LIN {X 0,Y 422.722,Z 380.789,A -85,B 0,C 180,E1 -10186.884,E2 -10186.884} C_VEL
LIN {X 0,Y 423.061,Z 367.924,A -85,B 0,C 180,E1 -10187.181,E2 -10187.181} C_VEL
LIN {X 0,Y 423.842,Z 291.469,A -85,B 0,C 180,E1 -10188.511,E2 -10188.511} C_VEL
LIN {X 0,Y 419.727,Z 266.585,A -85,B 0,C 180,E1 -10189.181,E2 -10189.181} C_VEL
LIN {X 0,Y 420.786,Z 249.269,A -85,B 0,C 180,E1 -10192.591,E2 -10192.591} C_VEL
LIN {X 0,Y 421.199,Z 242.855,A -85,B 0,C 180,E1 -10193.868,E2 -10193.868} C_VEL
LIN {X 0,Y 419.611,Z 233.827,A -85,B 0,C 180,E1 -10195.815,E2 -10195.815} C_VEL
LIN {X 0,Y 418.321,Z 227.378,A -85,B 0,C 180,E1 -10197.293,E2 -10197.293} C_VEL
LIN {X 0,Y 418.246,Z 227.386,A -85,B 0,C 180,E1 -10200.272,E2 -10200.272} C_VEL
LIN {X 0,Y 418.249,Z 227.389,A -85,B 0,C 180,E1 -10203.677,E2 -10203.677} C_VEL
LIN {X 0,Y 418.239,Z 227.391,A -85,B 0,C 180,E1 -10207.224,E2 -10207.224} C_VEL
LIN {X 0,Y 418.247,Z 227.385,A -85,B 0,C 180,E1 -10209.682,E2 -10209.682} C_VEL
LIN {X 0,Y 418.232,Z 227.384,A -85,B 0,C 180,E1 -10212.321,E2 -10212.321} C_VEL
LIN {X 0,Y 418.238,Z 227.388,A -85,B 0,C 180,E1 -10215.109,E2 -10215.109} C_VEL
LIN {X 0,Y 418.24,Z 227.383,A -85,B 0,C 180,E1 -10217.767,E2 -10217.767} C_VEL
LIN {X 0,Y 418.249,Z 227.385,A -85,B 0,C 180,E1 -10220.62,E2 -10220.62} C_VEL
LIN {X 0,Y 418.244,Z 227.382,A -85,B 0,C 180,E1 -10223.976,E2 -10223.976} C_VEL
LIN {X 0,Y 418.257,Z 227.386,A -85,B 0,C 180,E1 -10227.156,E2 -10227.156} C_VEL
LIN {X 0,Y 418.268,Z 227.385,A -85,B 0,C 180,E1 -10230.895,E2 -10230.895} C_VEL
LIN {X 0,Y 418.27,Z 227.38,A -85,B 0,C 180,E1 -10234.096,E2 -10234.096} C_VEL
LIN {X 0,Y 418.237,Z 227.385,A -85,B 0,C 180,E1 -10237.264,E2 -10237.264} C_VEL
LIN {X 0,Y 418.283,Z 227.379,A -85,B 0,C 180,E1 -10240.364,E2 -10240.364} C_VEL
LIN {X 0,Y 418.316,Z 227.377,A -85,B 0,C 180,E1 -10243.405,E2 -10243.405} C_VEL
LIN {X 0,Y 418.346,Z 227.372,A -85,B 0,C 180,E1 -10246.999,E2 -10246.999} C_VEL
LIN {X 0,Y 418.34,Z 227.369,A -85,B 0,C 180,E1 -10250.329,E2 -10250.329} C_VEL
LIN {X 0,Y 418.486,Z 227.355,A -85,B 0,C 180,E1 -10253.249,E2 -10253.249} C_VEL
LIN {X 0,Y 418.338,Z 227.371,A -85,B 0,C 180,E1 -10255.182,E2 -10255.182} C_VEL
LIN {X 0,Y 418.544,Z 227.347,A -85,B 0,C 180,E1 -10258.076,E2 -10258.076} C_VEL
LIN {X 0,Y 418.67,Z 227.325,A -85,B 0,C 180,E1 -10260,E2 -10260} C_VEL
LIN {X 0,Y 418.508,Z 227.352,A -85,B 0,C 180,E1 -10262.888,E2 -10262.888} C_VEL
LIN {X 0,Y 418.49,Z 227.357,A -85,B 0,C 180,E1 -10266.751,E2 -10266.751} C_VEL
LIN {X 0,Y 418.4,Z 227.365,A -85,B 0,C 180,E1 -10268.695,E2 -10268.695} C_VEL
LIN {X 0,Y 418.315,Z 227.371,A -85,B 0,C 180,E1 -10271.631,E2 -10271.631} C_VEL
LIN {X 0,Y 418.303,Z 227.38,A -85,B 0,C 180,E1 -10274.597,E2 -10274.597} C_VEL
LIN {X 0,Y 418.287,Z 227.378,A -85,B 0,C 180,E1 -10277.604,E2 -10277.604} C_VEL
LIN {X 0,Y 418.25,Z 227.387,A -85,B 0,C 180,E1 -10280.663,E2 -10280.663} C_VEL
LIN {X 0,Y 418.274,Z 227.379,A -85,B 0,C 180,E1 -10283.782,E2 -10283.782} C_VEL
LIN {X 0,Y 418.266,Z 227.384,A -85,B 0,C 180,E1 -10287.059,E2 -10287.059} C_VEL
LIN {X 0,Y 418.242,Z 227.386,A -85,B 0,C 180,E1 -10290.273,E2 -10290.273} C_VEL
LIN {X 0,Y 418.247,Z 227.388,A -85,B 0,C 180,E1 -10293.678,E2 -10293.678} C_VEL
LIN {X 0,Y 418.234,Z 227.388,A -85,B 0,C 180,E1 -10297.225,E2 -10297.225} C_VEL
LIN {X 0,Y 418.208,Z 227.393,A -85,B 0,C 180,E1 -10300.868,E2 -10300.868} C_VEL
LIN {X 0,Y 418.263,Z 227.487,A -85,B 0,C 180,E1 -10301.906,E2 -10301.906} C_VEL
LIN {X 0,Y 420.256,Z 237.548,A -85,B 0,C 180,E1 -10304.212,E2 -10304.212} C_VEL
LIN {X 0,Y 420.082,Z 245.787,A -85,B 0,C 180,E1 -10305.915,E2 -10305.915} C_VEL
LIN {X 0,Y 424.209,Z 265.63,A -85,B 0,C 180,E1 -10306.479,E2 -10306.479} C_VEL
LIN {X 0,Y 422.976,Z 353.633,A -85,B 0,C 180,E1 -10308.027,E2 -10308.027} C_VEL
LIN {X 0,Y 422.598,Z 366.879,A -85,B 0,C 180,E1 -10308.46,E2 -10308.46} C_VEL
LIN {X 0,Y 422.118,Z 378.903,A -85,B 0,C 180,E1 -10309.037,E2 -10309.037} C_VEL
LIN {X 0,Y 421.52,Z 390.055,A -85,B 0,C 180,E1 -10309.752,E2 -10309.752} C_VEL
LIN {X 0,Y 420.847,Z 400.567,A -85,B 0,C 180,E1 -10310.611,E2 -10310.611} C_VEL
LIN {X 0,Y 420.062,Z 411.702,A -85,B 0,C 180,E1 -10311.754,E2 -10311.754} C_VEL
LIN {X 0,Y 419.343,Z 420.671,A -85,B 0,C 180,E1 -10312.89,E2 -10312.89} C_VEL
LIN {X 0,Y 418.81,Z 428.099,A -85,B 0,C 180,E1 -10314.032,E2 -10314.032} C_VEL
LIN {X 0,Y 418.248,Z 435.582,A -85,B 0,C 180,E1 -10315.424,E2 -10315.424} C_VEL
LIN {X 0,Y 417.798,Z 441.651,A -85,B 0,C 180,E1 -10316.825,E2 -10316.825} C_VEL
LIN {X 0,Y 417.439,Z 447.432,A -85,B 0,C 180,E1 -10318.539,E2 -10318.539} C_VEL
LIN {X 0,Y 417.213,Z 451.593,A -85,B 0,C 180,E1 -10320.203,E2 -10320.203} C_VEL
LIN {X 0,Y 416.996,Z 454.414,A -85,B 0,C 180,E1 -10321.842,E2 -10321.842} C_VEL
LIN {X 0,Y 416.848,Z 455.921,A -85,B 0,C 180,E1 -10323.326,E2 -10323.326} C_VEL
LIN {X 0,Y 416.819,Z 456.5,A -85,B 0,C 180,E1 -10325.069,E2 -10325.069} C_VEL
LIN {X 0,Y 416.839,Z 456.196,A -85,B 0,C 180,E1 -10326.131,E2 -10326.131} C_VEL
LIN {X 0,Y 416.934,Z 454.562,A -85,B 0,C 180,E1 -10327.988,E2 -10327.988} C_VEL
LIN {X 0,Y 417.183,Z 451.479,A -85,B 0,C 180,E1 -10329.797,E2 -10329.797} C_VEL
LIN {X 0,Y 417.412,Z 447.619,A -85,B 0,C 180,E1 -10331.343,E2 -10331.343} C_VEL
LIN {X 0,Y 417.656,Z 442.562,A -85,B 0,C 180,E1 -10332.874,E2 -10332.874} C_VEL
LIN {X 0,Y 418.107,Z 436.133,A -85,B 0,C 180,E1 -10334.398,E2 -10334.398} C_VEL
LIN {X 0,Y 418.655,Z 428.087,A -85,B 0,C 180,E1 -10335.912,E2 -10335.912} C_VEL
LIN {X 0,Y 419.285,Z 419.45,A -85,B 0,C 180,E1 -10337.215,E2 -10337.215} C_VEL
LIN {X 0,Y 420.006,Z 409.662,A -85,B 0,C 180,E1 -10338.416,E2 -10338.416} C_VEL
LIN {X 0,Y 420.695,Z 398.721,A -85,B 0,C 180,E1 -10339.496,E2 -10339.496} C_VEL
LIN {X 0,Y 420.832,Z 397.065,A -85,B 0,C 180,E1 -10339.634,E2 -10339.634} C_VEL
LIN {X 0,Y 420.548,Z 392.07,A -85,B 0,C 180,E1 -10340.059,E2 -10340.059} C_VEL
LIN {X 0,Y 418.266,Z 383.781,A -85,B 0,C 180,E1 -10340.739,E2 -10340.739} C_VEL
LIN {X 0,Y 415.86,Z 375.215,A -85,B 0,C 180,E1 -10341.341,E2 -10341.341} C_VEL
LIN {X 0,Y 415.343,Z 369.734,A -85,B 0,C 180,E1 -10341.635,E2 -10341.635} C_VEL
LIN {X 0,Y 415.781,Z 356.858,A -85,B 0,C 180,E1 -10342.106,E2 -10342.106} C_VEL
LIN {X 0,Y 416.069,Z 340.665,A -85,B 0,C 180,E1 -10342.447,E2 -10342.447} C_VEL
LIN {X 0,Y 417.042,Z 266.429,A -85,B 0,C 180,E1 -10343.748,E2 -10343.748} C_VEL
LIN {X 0,Y 412.968,Z 245.698,A -85,B 0,C 180,E1 -10344.323,E2 -10344.323} C_VEL
LIN {X 0,Y 413.19,Z 239.008,A -85,B 0,C 180,E1 -10345.854,E2 -10345.854} C_VEL
LIN {X 0,Y 411.475,Z 228.232,A -85,B 0,C 180,E1 -10348.501,E2 -10348.501} C_VEL
LIN {X 0,Y 411.506,Z 228.226,A -85,B 0,C 180,E1 -10351.957,E2 -10351.957} C_VEL
LIN {X 0,Y 411.433,Z 228.236,A -85,B 0,C 180,E1 -10355.882,E2 -10355.882} C_VEL
LIN {X 0,Y 411.321,Z 228.246,A -85,B 0,C 180,E1 -10358.846,E2 -10358.846} C_VEL
LIN {X 0,Y 411.285,Z 228.255,A -85,B 0,C 180,E1 -10361.832,E2 -10361.832} C_VEL
LIN {X 0,Y 411.258,Z 228.254,A -85,B 0,C 180,E1 -10364.852,E2 -10364.852} C_VEL
LIN {X 0,Y 411.251,Z 228.259,A -85,B 0,C 180,E1 -10367.915,E2 -10367.915} C_VEL
LIN {X 0,Y 411.198,Z 228.262,A -85,B 0,C 180,E1 -10371.034,E2 -10371.034} C_VEL
LIN {X 0,Y 411.219,Z 228.261,A -85,B 0,C 180,E1 -10374.216,E2 -10374.216} C_VEL
LIN {X 0,Y 411.19,Z 228.266,A -85,B 0,C 180,E1 -10377.482,E2 -10377.482} C_VEL
LIN {X 0,Y 411.19,Z 228.263,A -85,B 0,C 180,E1 -10380.847,E2 -10380.847} C_VEL
LIN {X 0,Y 411.206,Z 228.263,A -85,B 0,C 180,E1 -10384.333,E2 -10384.333} C_VEL
LIN {X 0,Y 411.189,Z 228.266,A -85,B 0,C 180,E1 -10387.974,E2 -10387.974} C_VEL
LIN {X 0,Y 411.16,Z 228.268,A -85,B 0,C 180,E1 -10391.227,E2 -10391.227} C_VEL
LIN {X 0,Y 411.175,Z 228.267,A -85,B 0,C 180,E1 -10394.49,E2 -10394.49} C_VEL
LIN {X 0,Y 411.176,Z 228.267,A -85,B 0,C 180,E1 -10398.194,E2 -10398.194} C_VEL
LIN {X 0,Y 411.213,Z 228.261,A -85,B 0,C 180,E1 -10400.775,E2 -10400.775} C_VEL
LIN {X 0,Y 411.197,Z 228.265,A -85,B 0,C 180,E1 -10404.471,E2 -10404.471} C_VEL
LIN {X 0,Y 411.206,Z 228.262,A -85,B 0,C 180,E1 -10406.873,E2 -10406.873} C_VEL
LIN {X 0,Y 411.231,Z 228.26,A -85,B 0,C 180,E1 -10410.644,E2 -10410.644} C_VEL
LIN {X 0,Y 411.236,Z 228.261,A -85,B 0,C 180,E1 -10413.619,E2 -10413.619} C_VEL
LIN {X 0,Y 411.201,Z 228.263,A -85,B 0,C 180,E1 -10416.852,E2 -10416.852} C_VEL
LIN {X 0,Y 411.213,Z 228.263,A -85,B 0,C 180,E1 -10420.05,E2 -10420.05} C_VEL
LIN {X 0,Y 411.261,Z 228.255,A -85,B 0,C 180,E1 -10423.131,E2 -10423.131} C_VEL
LIN {X 0,Y 411.303,Z 228.25,A -85,B 0,C 180,E1 -10426.896,E2 -10426.896} C_VEL
LIN {X 0,Y 411.291,Z 228.254,A -85,B 0,C 180,E1 -10430.161,E2 -10430.161} C_VEL
LIN {X 0,Y 411.458,Z 228.23,A -85,B 0,C 180,E1 -10433.133,E2 -10433.133} C_VEL
LIN {X 0,Y 411.309,Z 228.249,A -85,B 0,C 180,E1 -10435.099,E2 -10435.099} C_VEL
LIN {X 0,Y 411.511,Z 228.226,A -85,B 0,C 180,E1 -10438.042,E2 -10438.042} C_VEL
LIN {X 0,Y 411.637,Z 228.21,A -85,B 0,C 180,E1 -10440,E2 -10440} C_VEL
LIN {X 0,Y 411.463,Z 228.23,A -85,B 0,C 180,E1 -10442.937,E2 -10442.937} C_VEL
LIN {X 0,Y 411.458,Z 228.231,A -85,B 0,C 180,E1 -10446.867,E2 -10446.867} C_VEL
LIN {X 0,Y 411.29,Z 228.253,A -85,B 0,C 180,E1 -10449.839,E2 -10449.839} C_VEL
LIN {X 0,Y 411.303,Z 228.25,A -85,B 0,C 180,E1 -10453.104,E2 -10453.104} C_VEL
LIN {X 0,Y 411.255,Z 228.256,A -85,B 0,C 180,E1 -10456.889,E2 -10456.889} C_VEL
LIN {X 0,Y 411.228,Z 228.261,A -85,B 0,C 180,E1 -10459.987,E2 -10459.987} C_VEL
LIN {X 0,Y 411.201,Z 228.262,A -85,B 0,C 180,E1 -10463.148,E2 -10463.148} C_VEL
LIN {X 0,Y 411.235,Z 228.262,A -85,B 0,C 180,E1 -10466.381,E2 -10466.381} C_VEL
LIN {X 0,Y 411.198,Z 228.263,A -85,B 0,C 180,E1 -10469.713,E2 -10469.713} C_VEL
LIN {X 0,Y 411.204,Z 228.261,A -85,B 0,C 180,E1 -10473.156,E2 -10473.156} C_VEL
LIN {X 0,Y 411.191,Z 228.268,A -85,B 0,C 180,E1 -10476.553,E2 -10476.553} C_VEL
LIN {X 0,Y 411.211,Z 228.261,A -85,B 0,C 180,E1 -10479.728,E2 -10479.728} C_VEL
LIN {X 0,Y 411.172,Z 228.265,A -85,B 0,C 180,E1 -10483.134,E2 -10483.134} C_VEL
LIN {X 0,Y 411.167,Z 228.267,A -85,B 0,C 180,E1 -10485.881,E2 -10485.881} C_VEL
LIN {X 0,Y 411.163,Z 228.269,A -85,B 0,C 180,E1 -10488.772,E2 -10488.772} C_VEL
LIN {X 0,Y 411.205,Z 228.261,A -85,B 0,C 180,E1 -10491.832,E2 -10491.832} C_VEL
LIN {X 0,Y 411.21,Z 228.26,A -85,B 0,C 180,E1 -10495.122,E2 -10495.122} C_VEL
LIN {X 0,Y 411.166,Z 228.267,A -85,B 0,C 180,E1 -10498.003,E2 -10498.003} C_VEL
LIN {X 0,Y 411.218,Z 228.262,A -85,B 0,C 180,E1 -10501.41,E2 -10501.41} C_VEL
LIN {X 0,Y 411.302,Z 228.423,A -85,B 0,C 180,E1 -10502.526,E2 -10502.526} C_VEL
LIN {X 0,Y 413.808,Z 241.239,A -85,B 0,C 180,E1 -10505.412,E2 -10505.412} C_VEL
LIN {X 0,Y 414.227,Z 245.195,A -85,B 0,C 180,E1 -10506.264,E2 -10506.264} C_VEL
LIN {X 0,Y 413.042,Z 262.161,A -85,B 0,C 180,E1 -10509.718,E2 -10509.718} C_VEL
LIN {X 0,Y 412.704,Z 267.045,A -85,B 0,C 180,E1 -10510.704,E2 -10510.704} C_VEL
LIN {X 0,Y 416.828,Z 293.741,A -85,B 0,C 180,E1 -10511.378,E2 -10511.378} C_VEL
LIN {X 0,Y 415.814,Z 375.201,A -85,B 0,C 180,E1 -10512.828,E2 -10512.828} C_VEL
LIN {X 0,Y 415.314,Z 388.414,A -85,B 0,C 180,E1 -10513.25,E2 -10513.25} C_VEL
LIN {X 0,Y 414.714,Z 400.568,A -85,B 0,C 180,E1 -10513.826,E2 -10513.826} C_VEL
LIN {X 0,Y 413.928,Z 412.845,A -85,B 0,C 180,E1 -10514.616,E2 -10514.616} C_VEL
LIN {X 0,Y 413.184,Z 424.428,A -85,B 0,C 180,E1 -10515.593,E2 -10515.593} C_VEL
LIN {X 0,Y 412.456,Z 434.918,A -85,B 0,C 180,E1 -10516.701,E2 -10516.701} C_VEL
LIN {X 0,Y 411.765,Z 444.323,A -85,B 0,C 180,E1 -10517.932,E2 -10517.932} C_VEL
LIN {X 0,Y 411.017,Z 453.403,A -85,B 0,C 180,E1 -10519.408,E2 -10519.408} C_VEL
LIN {X 0,Y 410.572,Z 460.724,A -85,B 0,C 180,E1 -10520.89,E2 -10520.89} C_VEL
LIN {X 0,Y 410.292,Z 465.675,A -85,B 0,C 180,E1 -10522.124,E2 -10522.124} C_VEL
LIN {X 0,Y 410.058,Z 470.92,A -85,B 0,C 180,E1 -10523.755,E2 -10523.755} C_VEL
LIN {X 0,Y 410.018,Z 474.159,A -85,B 0,C 180,E1 -10525.084,E2 -10525.084} C_VEL
LIN {X 0,Y 409.931,Z 476.057,A -85,B 0,C 180,E1 -10526.068,E2 -10526.068} C_VEL
LIN {X 0,Y 409.926,Z 477.497,A -85,B 0,C 180,E1 -10527.052,E2 -10527.052} C_VEL
LIN {X 0,Y 409.966,Z 478.515,A -85,B 0,C 180,E1 -10528.035,E2 -10528.035} C_VEL
LIN {X 0,Y 409.927,Z 479.378,A -85,B 0,C 180,E1 -10530,E2 -10530} C_VEL
LIN {X 0,Y 409.936,Z 479.189,A -85,B 0,C 180,E1 -10530.982,E2 -10530.982} C_VEL
LIN {X 0,Y 409.966,Z 478.591,A -85,B 0,C 180,E1 -10531.965,E2 -10531.965} C_VEL
LIN {X 0,Y 409.931,Z 476.216,A -85,B 0,C 180,E1 -10533.932,E2 -10533.932} C_VEL
LIN {X 0,Y 410.017,Z 473.291,A -85,B 0,C 180,E1 -10535.41,E2 -10535.41} C_VEL
LIN {X 0,Y 410.166,Z 469.333,A -85,B 0,C 180,E1 -10536.889,E2 -10536.889} C_VEL
LIN {X 0,Y 410.477,Z 463.255,A -85,B 0,C 180,E1 -10538.616,E2 -10538.616} C_VEL
LIN {X 0,Y 410.919,Z 456.598,A -85,B 0,C 180,E1 -10540.097,E2 -10540.097} C_VEL
LIN {X 0,Y 411.535,Z 448.339,A -85,B 0,C 180,E1 -10541.576,E2 -10541.576} C_VEL
LIN {X 0,Y 412.255,Z 439.9,A -85,B 0,C 180,E1 -10542.804,E2 -10542.804} C_VEL
LIN {X 0,Y 412.93,Z 430.53,A -85,B 0,C 180,E1 -10543.925,E2 -10543.925} C_VEL
LIN {X 0,Y 413.71,Z 419.198,A -85,B 0,C 180,E1 -10545.015,E2 -10545.015} C_VEL
LIN {X 0,Y 414.509,Z 407.954,A -85,B 0,C 180,E1 -10545.867,E2 -10545.867} C_VEL
LIN {X 0,Y 415.235,Z 396.565,A -85,B 0,C 180,E1 -10546.532,E2 -10546.532} C_VEL
LIN {X 0,Y 415.827,Z 383.626,A -85,B 0,C 180,E1 -10547.077,E2 -10547.077} C_VEL
LIN {X 0,Y 416.261,Z 369.921,A -85,B 0,C 180,E1 -10547.439,E2 -10547.439} C_VEL
LIN {X 0,Y 417.167,Z 292.496,A -85,B 0,C 180,E1 -10548.811,E2 -10548.811} C_VEL
LIN {X 0,Y 412.834,Z 266.4,A -85,B 0,C 180,E1 -10549.526,E2 -10549.526} C_VEL
LIN {X 0,Y 414.044,Z 247.988,A -85,B 0,C 180,E1 -10553.217,E2 -10553.217} C_VEL
LIN {X 0,Y 414.101,Z 242.72,A -85,B 0,C 180,E1 -10554.303,E2 -10554.303} C_VEL
LIN {X 0,Y 411.579,Z 229.792,A -85,B 0,C 180,E1 -10557.183,E2 -10557.183} C_VEL
LIN {X 0,Y 411.304,Z 228.252,A -85,B 0,C 180,E1 -10557.543,E2 -10557.543} C_VEL
LIN {X 0,Y 411.191,Z 228.267,A -85,B 0,C 180,E1 -10560.847,E2 -10560.847} C_VEL
LIN {X 0,Y 411.206,Z 228.263,A -85,B 0,C 180,E1 -10564.333,E2 -10564.333} C_VEL
LIN {X 0,Y 411.193,Z 228.263,A -85,B 0,C 180,E1 -10567.974,E2 -10567.974} C_VEL
LIN {X 0,Y 411.165,Z 228.272,A -85,B 0,C 180,E1 -10571.228,E2 -10571.228} C_VEL
LIN {X 0,Y 411.18,Z 228.266,A -85,B 0,C 180,E1 -10574.49,E2 -10574.49} C_VEL
LIN {X 0,Y 411.177,Z 228.261,A -85,B 0,C 180,E1 -10578.194,E2 -10578.194} C_VEL
LIN {X 0,Y 411.214,Z 228.263,A -85,B 0,C 180,E1 -10580.775,E2 -10580.775} C_VEL
LIN {X 0,Y 411.198,Z 228.26,A -85,B 0,C 180,E1 -10584.471,E2 -10584.471} C_VEL
LIN {X 0,Y 411.207,Z 228.264,A -85,B 0,C 180,E1 -10586.873,E2 -10586.873} C_VEL
LIN {X 0,Y 411.232,Z 228.258,A -85,B 0,C 180,E1 -10590.644,E2 -10590.644} C_VEL
LIN {X 0,Y 411.237,Z 228.257,A -85,B 0,C 180,E1 -10593.619,E2 -10593.619} C_VEL
LIN {X 0,Y 411.203,Z 228.26,A -85,B 0,C 180,E1 -10596.852,E2 -10596.852} C_VEL
LIN {X 0,Y 411.214,Z 228.259,A -85,B 0,C 180,E1 -10600.05,E2 -10600.05} C_VEL
LIN {X 0,Y 411.262,Z 228.259,A -85,B 0,C 180,E1 -10603.131,E2 -10603.131} C_VEL
LIN {X 0,Y 411.305,Z 228.247,A -85,B 0,C 180,E1 -10606.896,E2 -10606.896} C_VEL
LIN {X 0,Y 411.292,Z 228.246,A -85,B 0,C 180,E1 -10610.161,E2 -10610.161} C_VEL
LIN {X 0,Y 411.451,Z 228.233,A -85,B 0,C 180,E1 -10613.133,E2 -10613.133} C_VEL
LIN {X 0,Y 411.309,Z 228.246,A -85,B 0,C 180,E1 -10615.099,E2 -10615.099} C_VEL
LIN {X 0,Y 411.513,Z 228.222,A -85,B 0,C 180,E1 -10618.043,E2 -10618.043} C_VEL
LIN {X 0,Y 411.639,Z 228.2,A -85,B 0,C 180,E1 -10620,E2 -10620} C_VEL
LIN {X 0,Y 411.463,Z 228.229,A -85,B 0,C 180,E1 -10622.937,E2 -10622.937} C_VEL
LIN {X 0,Y 411.458,Z 228.231,A -85,B 0,C 180,E1 -10626.867,E2 -10626.867} C_VEL
LIN {X 0,Y 411.354,Z 228.244,A -85,B 0,C 180,E1 -10628.845,E2 -10628.845} C_VEL
LIN {X 0,Y 411.283,Z 228.247,A -85,B 0,C 180,E1 -10631.833,E2 -10631.833} C_VEL
LIN {X 0,Y 411.26,Z 228.255,A -85,B 0,C 180,E1 -10634.853,E2 -10634.853} C_VEL
LIN {X 0,Y 411.252,Z 228.255,A -85,B 0,C 180,E1 -10637.915,E2 -10637.915} C_VEL
LIN {X 0,Y 411.196,Z 228.263,A -85,B 0,C 180,E1 -10641.034,E2 -10641.034} C_VEL
LIN {X 0,Y 411.212,Z 228.261,A -85,B 0,C 180,E1 -10644.217,E2 -10644.217} C_VEL
LIN {X 0,Y 411.207,Z 228.261,A -85,B 0,C 180,E1 -10647.482,E2 -10647.482} C_VEL
LIN {X 0,Y 411.189,Z 228.266,A -85,B 0,C 180,E1 -10650.848,E2 -10650.848} C_VEL
LIN {X 0,Y 411.204,Z 228.267,A -85,B 0,C 180,E1 -10654.334,E2 -10654.334} C_VEL
LIN {X 0,Y 411.183,Z 228.269,A -85,B 0,C 180,E1 -10657.975,E2 -10657.975} C_VEL
LIN {X 0,Y 411.218,Z 228.345,A -85,B 0,C 180,E1 -10661.619,E2 -10661.619} C_VEL
LIN {X 0,Y 413.367,Z 239.371,A -85,B 0,C 180,E1 -10664.193,E2 -10664.193} C_VEL
LIN {X 0,Y 413.217,Z 245.893,A -85,B 0,C 180,E1 -10665.565,E2 -10665.565} C_VEL
LIN {X 0,Y 417.588,Z 267.363,A -85,B 0,C 180,E1 -10666.186,E2 -10666.186} C_VEL
LIN {X 0,Y 416.254,Z 353.529,A -85,B 0,C 180,E1 -10667.724,E2 -10667.724} C_VEL
LIN {X 0,Y 415.848,Z 366.678,A -85,B 0,C 180,E1 -10668.155,E2 -10668.155} C_VEL
LIN {X 0,Y 415.301,Z 379.497,A -85,B 0,C 180,E1 -10668.779,E2 -10668.779} C_VEL
LIN {X 0,Y 414.641,Z 391.093,A -85,B 0,C 180,E1 -10669.547,E2 -10669.547} C_VEL
LIN {X 0,Y 413.794,Z 403.296,A -85,B 0,C 180,E1 -10670.596,E2 -10670.596} C_VEL
LIN {X 0,Y 413.032,Z 413.572,A -85,B 0,C 180,E1 -10671.712,E2 -10671.712} C_VEL
LIN {X 0,Y 412.262,Z 423.509,A -85,B 0,C 180,E1 -10673.065,E2 -10673.065} C_VEL
LIN {X 0,Y 411.542,Z 432.054,A -85,B 0,C 180,E1 -10674.506,E2 -10674.506} C_VEL
LIN {X 0,Y 410.998,Z 438.911,A -85,B 0,C 180,E1 -10675.943,E2 -10675.943} C_VEL
LIN {X 0,Y 410.582,Z 444.679,A -85,B 0,C 180,E1 -10677.463,E2 -10677.463} C_VEL
LIN {X 0,Y 410.291,Z 449.42,A -85,B 0,C 180,E1 -10679.078,E2 -10679.078} C_VEL
LIN {X 0,Y 410.043,Z 453.356,A -85,B 0,C 180,E1 -10680.942,E2 -10680.942} C_VEL
LIN {X 0,Y 409.833,Z 455.36,A -85,B 0,C 180,E1 -10682.419,E2 -10682.419} C_VEL
LIN {X 0,Y 409.74,Z 456.267,A -85,B 0,C 180,E1 -10683.515,E2 -10683.515} C_VEL
LIN {X 0,Y 409.724,Z 456.64,A -85,B 0,C 180,E1 -10685.383,E2 -10685.383} C_VEL
LIN {X 0,Y 409.762,Z 456.014,A -85,B 0,C 180,E1 -10686.766,E2 -10686.766} C_VEL
LIN {X 0,Y 409.838,Z 454.975,A -85,B 0,C 180,E1 -10687.836,E2 -10687.836} C_VEL
LIN {X 0,Y 410.031,Z 452.536,A -85,B 0,C 180,E1 -10689.429,E2 -10689.429} C_VEL
LIN {X 0,Y 410.272,Z 448.998,A -85,B 0,C 180,E1 -10691.006,E2 -10691.006} C_VEL
LIN {X 0,Y 410.527,Z 444.298,A -85,B 0,C 180,E1 -10692.567,E2 -10692.567} C_VEL
LIN {X 0,Y 410.933,Z 438.259,A -85,B 0,C 180,E1 -10694.119,E2 -10694.119} C_VEL
LIN {X 0,Y 411.494,Z 430.659,A -85,B 0,C 180,E1 -10695.662,E2 -10695.662} C_VEL
LIN {X 0,Y 412.143,Z 422.261,A -85,B 0,C 180,E1 -10697.036,E2 -10697.036} C_VEL
LIN {X 0,Y 412.867,Z 412.405,A -85,B 0,C 180,E1 -10698.338,E2 -10698.338} C_VEL
LIN {X 0,Y 413.624,Z 401.995,A -85,B 0,C 180,E1 -10699.439,E2 -10699.439} C_VEL
LIN {X 0,Y 414.378,Z 391.15,A -85,B 0,C 180,E1 -10700.358,E2 -10700.358} C_VEL
LIN {X 0,Y 415.01,Z 378.845,A -85,B 0,C 180,E1 -10701.172,E2 -10701.172} C_VEL
LIN {X 0,Y 415.343,Z 369.734,A -85,B 0,C 180,E1 -10701.635,E2 -10701.635} C_VEL
LIN {X 0,Y 414.883,Z 364.151,A -85,B 0,C 180,E1 -10701.896,E2 -10701.896} C_VEL
LIN {X 0,Y 412.386,Z 354.998,A -85,B 0,C 180,E1 -10702.298,E2 -10702.298} C_VEL
LIN {X 0,Y 409.847,Z 345.704,A -85,B 0,C 180,E1 -10702.618,E2 -10702.618} C_VEL
LIN {X 0,Y 409.307,Z 339.901,A -85,B 0,C 180,E1 -10702.746,E2 -10702.746} C_VEL
LIN {X 0,Y 410.232,Z 267.175,A -85,B 0,C 180,E1 -10704.044,E2 -10704.044} C_VEL
LIN {X 0,Y 406.065,Z 245.83,A -85,B 0,C 180,E1 -10704.659,E2 -10704.659} C_VEL
LIN {X 0,Y 406.177,Z 239.949,A -85,B 0,C 180,E1 -10706.031,E2 -10706.031} C_VEL
LIN {X 0,Y 404.599,Z 229.943,A -85,B 0,C 180,E1 -10708.507,E2 -10708.507} C_VEL
LIN {X 0,Y 404.422,Z 229.11,A -85,B 0,C 180,E1 -10708.755,E2 -10708.755} C_VEL
LIN {X 0,Y 404.475,Z 229.102,A -85,B 0,C 180,E1 -10711.991,E2 -10711.991} C_VEL
LIN {X 0,Y 404.381,Z 229.114,A -85,B 0,C 180,E1 -10715.985,E2 -10715.985} C_VEL
LIN {X 0,Y 404.268,Z 229.125,A -85,B 0,C 180,E1 -10719.001,E2 -10719.001} C_VEL
LIN {X 0,Y 404.258,Z 229.129,A -85,B 0,C 180,E1 -10722.041,E2 -10722.041} C_VEL
LIN {X 0,Y 404.204,Z 229.133,A -85,B 0,C 180,E1 -10725.118,E2 -10725.118} C_VEL
LIN {X 0,Y 404.209,Z 229.134,A -85,B 0,C 180,E1 -10728.238,E2 -10728.238} C_VEL
LIN {X 0,Y 404.141,Z 229.143,A -85,B 0,C 180,E1 -10731.419,E2 -10731.419} C_VEL
LIN {X 0,Y 404.168,Z 229.138,A -85,B 0,C 180,E1 -10734.666,E2 -10734.666} C_VEL
LIN {X 0,Y 404.132,Z 229.145,A -85,B 0,C 180,E1 -10738.004,E2 -10738.004} C_VEL
LIN {X 0,Y 404.145,Z 229.142,A -85,B 0,C 180,E1 -10740.285,E2 -10740.285} C_VEL
LIN {X 0,Y 404.145,Z 229.145,A -85,B 0,C 180,E1 -10743.812,E2 -10743.812} C_VEL
LIN {X 0,Y 404.135,Z 229.142,A -85,B 0,C 180,E1 -10746.874,E2 -10746.874} C_VEL
LIN {X 0,Y 404.147,Z 229.143,A -85,B 0,C 180,E1 -10750.08,E2 -10750.08} C_VEL
LIN {X 0,Y 404.15,Z 229.14,A -85,B 0,C 180,E1 -10753.083,E2 -10753.083} C_VEL
LIN {X 0,Y 404.147,Z 229.144,A -85,B 0,C 180,E1 -10755.926,E2 -10755.926} C_VEL
LIN {X 0,Y 404.117,Z 229.145,A -85,B 0,C 180,E1 -10758.634,E2 -10758.634} C_VEL
LIN {X 0,Y 404.151,Z 229.142,A -85,B 0,C 180,E1 -10761.492,E2 -10761.492} C_VEL
LIN {X 0,Y 404.184,Z 229.136,A -85,B 0,C 180,E1 -10764.984,E2 -10764.984} C_VEL
LIN {X 0,Y 404.14,Z 229.143,A -85,B 0,C 180,E1 -10768.553,E2 -10768.553} C_VEL
LIN {X 0,Y 404.193,Z 229.138,A -85,B 0,C 180,E1 -10772,E2 -10772} C_VEL
LIN {X 0,Y 404.175,Z 229.138,A -85,B 0,C 180,E1 -10775.334,E2 -10775.334} C_VEL
LIN {X 0,Y 404.137,Z 229.144,A -85,B 0,C 180,E1 -10778.58,E2 -10778.58} C_VEL
LIN {X 0,Y 404.208,Z 229.137,A -85,B 0,C 180,E1 -10781.762,E2 -10781.762} C_VEL
LIN {X 0,Y 404.204,Z 229.134,A -85,B 0,C 180,E1 -10784.882,E2 -10784.882} C_VEL
LIN {X 0,Y 404.254,Z 229.13,A -85,B 0,C 180,E1 -10787.958,E2 -10787.958} C_VEL
LIN {X 0,Y 404.431,Z 229.108,A -85,B 0,C 180,E1 -10792.099,E2 -10792.099} C_VEL
LIN {X 0,Y 404.422,Z 229.109,A -85,B 0,C 180,E1 -10794.015,E2 -10794.015} C_VEL
LIN {X 0,Y 404.48,Z 229.102,A -85,B 0,C 180,E1 -10798.008,E2 -10798.008} C_VEL
LIN {X 0,Y 404.607,Z 229.086,A -85,B 0,C 180,E1 -10800,E2 -10800} C_VEL
LIN {X 0,Y 404.42,Z 229.107,A -85,B 0,C 180,E1 -10802.988,E2 -10802.988} C_VEL
LIN {X 0,Y 404.409,Z 229.108,A -85,B 0,C 180,E1 -10806.987,E2 -10806.987} C_VEL
LIN {X 0,Y 404.255,Z 229.13,A -85,B 0,C 180,E1 -10810.012,E2 -10810.012} C_VEL
LIN {X 0,Y 404.264,Z 229.126,A -85,B 0,C 180,E1 -10813.211,E2 -10813.211} C_VEL
LIN {X 0,Y 404.213,Z 229.133,A -85,B 0,C 180,E1 -10817.007,E2 -10817.007} C_VEL
LIN {X 0,Y 404.161,Z 229.143,A -85,B 0,C 180,E1 -10820.352,E2 -10820.352} C_VEL
LIN {X 0,Y 404.167,Z 229.138,A -85,B 0,C 180,E1 -10823.575,E2 -10823.575} C_VEL
LIN {X 0,Y 404.181,Z 229.138,A -85,B 0,C 180,E1 -10825.767,E2 -10825.767} C_VEL
LIN {X 0,Y 404.193,Z 229.137,A -85,B 0,C 180,E1 -10828,E2 -10828} C_VEL
LIN {X 0,Y 404.137,Z 229.142,A -85,B 0,C 180,E1 -10831.558,E2 -10831.558} C_VEL
LIN {X 0,Y 404.183,Z 229.136,A -85,B 0,C 180,E1 -10835.016,E2 -10835.016} C_VEL
LIN {X 0,Y 404.152,Z 229.142,A -85,B 0,C 180,E1 -10838.757,E2 -10838.757} C_VEL
LIN {X 0,Y 404.121,Z 229.143,A -85,B 0,C 180,E1 -10841.6,E2 -10841.6} C_VEL
LIN {X 0,Y 404.144,Z 229.146,A -85,B 0,C 180,E1 -10844.522,E2 -10844.522} C_VEL
LIN {X 0,Y 404.136,Z 229.141,A -85,B 0,C 180,E1 -10847.296,E2 -10847.296} C_VEL
LIN {X 0,Y 404.168,Z 229.139,A -85,B 0,C 180,E1 -10849.956,E2 -10849.956} C_VEL
LIN {X 0,Y 404.135,Z 229.141,A -85,B 0,C 180,E1 -10853.126,E2 -10853.126} C_VEL
LIN {X 0,Y 404.145,Z 229.143,A -85,B 0,C 180,E1 -10856.188,E2 -10856.188} C_VEL
LIN {X 0,Y 404.146,Z 229.143,A -85,B 0,C 180,E1 -10859.715,E2 -10859.715} C_VEL
LIN {X 0,Y 404.264,Z 229.217,A -85,B 0,C 180,E1 -10862.245,E2 -10862.245} C_VEL
LIN {X 0,Y 406.786,Z 242.234,A -85,B 0,C 180,E1 -10865.231,E2 -10865.231} C_VEL
LIN {X 0,Y 407.267,Z 246.402,A -85,B 0,C 180,E1 -10866.148,E2 -10866.148} C_VEL
LIN {X 0,Y 406.095,Z 262.277,A -85,B 0,C 180,E1 -10869.437,E2 -10869.437} C_VEL
LIN {X 0,Y 405.773,Z 266.848,A -85,B 0,C 180,E1 -10870.376,E2 -10870.376} C_VEL
LIN {X 0,Y 410.051,Z 293.907,A -85,B 0,C 180,E1 -10871.08,E2 -10871.08} C_VEL
LIN {X 0,Y 408.98,Z 375.579,A -85,B 0,C 180,E1 -10872.564,E2 -10872.564} C_VEL
LIN {X 0,Y 408.428,Z 389.361,A -85,B 0,C 180,E1 -10873.023,E2 -10873.023} C_VEL
LIN {X 0,Y 407.826,Z 401.221,A -85,B 0,C 180,E1 -10873.609,E2 -10873.609} C_VEL
LIN {X 0,Y 407.082,Z 412.453,A -85,B 0,C 180,E1 -10874.351,E2 -10874.351} C_VEL
LIN {X 0,Y 406.254,Z 424.492,A -85,B 0,C 180,E1 -10875.383,E2 -10875.383} C_VEL
LIN {X 0,Y 405.53,Z 434.59,A -85,B 0,C 180,E1 -10876.47,E2 -10876.47} C_VEL
LIN {X 0,Y 404.794,Z 444.027,A -85,B 0,C 180,E1 -10877.721,E2 -10877.721} C_VEL
LIN {X 0,Y 403.999,Z 453.126,A -85,B 0,C 180,E1 -10879.222,E2 -10879.222} C_VEL
LIN {X 0,Y 403.517,Z 460.461,A -85,B 0,C 180,E1 -10880.729,E2 -10880.729} C_VEL
LIN {X 0,Y 403.23,Z 465.425,A -85,B 0,C 180,E1 -10881.985,E2 -10881.985} C_VEL
LIN {X 0,Y 402.979,Z 471.026,A -85,B 0,C 180,E1 -10883.768,E2 -10883.768} C_VEL
LIN {X 0,Y 402.93,Z 473.933,A -85,B 0,C 180,E1 -10884.997,E2 -10884.997} C_VEL
LIN {X 0,Y 402.852,Z 475.836,A -85,B 0,C 180,E1 -10885.999,E2 -10885.999} C_VEL
LIN {X 0,Y 402.825,Z 477.285,A -85,B 0,C 180,E1 -10887,E2 -10887} C_VEL
LIN {X 0,Y 402.864,Z 478.308,A -85,B 0,C 180,E1 -10888.001,E2 -10888.001} C_VEL
LIN {X 0,Y 402.862,Z 478.938,A -85,B 0,C 180,E1 -10889.001,E2 -10889.001} C_VEL
LIN {X 0,Y 402.852,Z 479.18,A -85,B 0,C 180,E1 -10890,E2 -10890} C_VEL
LIN {X 0,Y 402.863,Z 478.998,A -85,B 0,C 180,E1 -10891,E2 -10891} C_VEL
LIN {X 0,Y 402.864,Z 478.404,A -85,B 0,C 180,E1 -10892,E2 -10892} C_VEL
LIN {X 0,Y 402.852,Z 476.036,A -85,B 0,C 180,E1 -10894.002,E2 -10894.002} C_VEL
LIN {X 0,Y 402.915,Z 473.117,A -85,B 0,C 180,E1 -10895.505,E2 -10895.505} C_VEL
LIN {X 0,Y 403.08,Z 469.166,A -85,B 0,C 180,E1 -10897.011,E2 -10897.011} C_VEL
LIN {X 0,Y 403.363,Z 464.079,A -85,B 0,C 180,E1 -10898.517,E2 -10898.517} C_VEL
LIN {X 0,Y 403.808,Z 457.69,A -85,B 0,C 180,E1 -10900.023,E2 -10900.023} C_VEL
LIN {X 0,Y 404.401,Z 449.698,A -85,B 0,C 180,E1 -10901.529,E2 -10901.529} C_VEL
LIN {X 0,Y 405.308,Z 439.776,A -85,B 0,C 180,E1 -10903.028,E2 -10903.028} C_VEL
LIN {X 0,Y 406.02,Z 429.895,A -85,B 0,C 180,E1 -10904.226,E2 -10904.226} C_VEL
LIN {X 0,Y 406.857,Z 419.14,A -85,B 0,C 180,E1 -10905.274,E2 -10905.274} C_VEL
LIN {X 0,Y 407.694,Z 407.941,A -85,B 0,C 180,E1 -10906.139,E2 -10906.139} C_VEL
LIN {X 0,Y 408.529,Z 395.407,A -85,B 0,C 180,E1 -10906.876,E2 -10906.876} C_VEL
LIN {X 0,Y 409.117,Z 382.04,A -85,B 0,C 180,E1 -10907.431,E2 -10907.431} C_VEL
LIN {X 0,Y 409.552,Z 368.972,A -85,B 0,C 180,E1 -10907.766,E2 -10907.766} C_VEL
LIN {X 0,Y 410.454,Z 293.26,A -85,B 0,C 180,E1 -10909.13,E2 -10909.13} C_VEL
LIN {X 0,Y 405.953,Z 266.262,A -85,B 0,C 180,E1 -10909.874,E2 -10909.874} C_VEL
LIN {X 0,Y 407.128,Z 249.014,A -85,B 0,C 180,E1 -10913.393,E2 -10913.393} C_VEL
LIN {X 0,Y 407.336,Z 245.679,A -85,B 0,C 180,E1 -10914.082,E2 -10914.082} C_VEL
LIN {X 0,Y 406.009,Z 237.858,A -85,B 0,C 180,E1 -10915.826,E2 -10915.826} C_VEL
LIN {X 0,Y 404.252,Z 229.132,A -85,B 0,C 180,E1 -10917.859,E2 -10917.859} C_VEL
LIN {X 0,Y 404.141,Z 229.147,A -85,B 0,C 180,E1 -10921.558,E2 -10921.558} C_VEL
LIN {X 0,Y 404.185,Z 229.141,A -85,B 0,C 180,E1 -10925.016,E2 -10925.016} C_VEL
LIN {X 0,Y 404.153,Z 229.141,A -85,B 0,C 180,E1 -10928.757,E2 -10928.757} C_VEL
LIN {X 0,Y 404.124,Z 229.145,A -85,B 0,C 180,E1 -10931.6,E2 -10931.6} C_VEL
LIN {X 0,Y 404.149,Z 229.142,A -85,B 0,C 180,E1 -10934.522,E2 -10934.522} C_VEL
LIN {X 0,Y 404.136,Z 229.145,A -85,B 0,C 180,E1 -10937.295,E2 -10937.295} C_VEL
LIN {X 0,Y 404.169,Z 229.138,A -85,B 0,C 180,E1 -10939.955,E2 -10939.955} C_VEL
LIN {X 0,Y 404.136,Z 229.147,A -85,B 0,C 180,E1 -10943.125,E2 -10943.125} C_VEL
LIN {X 0,Y 404.145,Z 229.139,A -85,B 0,C 180,E1 -10946.188,E2 -10946.188} C_VEL
LIN {X 0,Y 404.145,Z 229.14,A -85,B 0,C 180,E1 -10949.715,E2 -10949.715} C_VEL
LIN {X 0,Y 404.195,Z 229.133,A -85,B 0,C 180,E1 -10953.123,E2 -10953.123} C_VEL
LIN {X 0,Y 404.177,Z 229.138,A -85,B 0,C 180,E1 -10955.334,E2 -10955.334} C_VEL
LIN {X 0,Y 404.138,Z 229.141,A -85,B 0,C 180,E1 -10958.581,E2 -10958.581} C_VEL
LIN {X 0,Y 404.209,Z 229.128,A -85,B 0,C 180,E1 -10961.762,E2 -10961.762} C_VEL
LIN {X 0,Y 404.206,Z 229.133,A -85,B 0,C 180,E1 -10964.882,E2 -10964.882} C_VEL
LIN {X 0,Y 404.256,Z 229.125,A -85,B 0,C 180,E1 -10967.959,E2 -10967.959} C_VEL
LIN {X 0,Y 404.404,Z 229.106,A -85,B 0,C 180,E1 -10972.129,E2 -10972.129} C_VEL
LIN {X 0,Y 404.418,Z 229.104,A -85,B 0,C 180,E1 -10974.015,E2 -10974.015} C_VEL
LIN {X 0,Y 404.482,Z 229.098,A -85,B 0,C 180,E1 -10978.009,E2 -10978.009} C_VEL
LIN {X 0,Y 404.609,Z 229.076,A -85,B 0,C 180,E1 -10980,E2 -10980} C_VEL
LIN {X 0,Y 404.42,Z 229.105,A -85,B 0,C 180,E1 -10982.989,E2 -10982.989} C_VEL
LIN {X 0,Y 404.409,Z 229.107,A -85,B 0,C 180,E1 -10986.987,E2 -10986.987} C_VEL
LIN {X 0,Y 404.258,Z 229.127,A -85,B 0,C 180,E1 -10990.012,E2 -10990.012} C_VEL
LIN {X 0,Y 404.266,Z 229.127,A -85,B 0,C 180,E1 -10993.212,E2 -10993.212} C_VEL
LIN {X 0,Y 404.215,Z 229.134,A -85,B 0,C 180,E1 -10997.007,E2 -10997.007} C_VEL
LIN {X 0,Y 404.163,Z 229.142,A -85,B 0,C 180,E1 -11000.352,E2 -11000.352} C_VEL
LIN {X 0,Y 404.16,Z 229.137,A -85,B 0,C 180,E1 -11003.575,E2 -11003.575} C_VEL
LIN {X 0,Y 404.151,Z 229.144,A -85,B 0,C 180,E1 -11006.88,E2 -11006.88} C_VEL
LIN {X 0,Y 404.144,Z 229.142,A -85,B 0,C 180,E1 -11010.285,E2 -11010.285} C_VEL
LIN {X 0,Y 404.144,Z 229.145,A -85,B 0,C 180,E1 -11013.813,E2 -11013.813} C_VEL
LIN {X 0,Y 404.132,Z 229.146,A -85,B 0,C 180,E1 -11016.874,E2 -11016.874} C_VEL
LIN {X 0,Y 404.117,Z 229.149,A -85,B 0,C 180,E1 -11020.075,E2 -11020.075} C_VEL
LIN {X 0,Y 404.164,Z 229.194,A -85,B 0,C 180,E1 -11021.318,E2 -11021.318} C_VEL
LIN {X 0,Y 406.437,Z 240.61,A -85,B 0,C 180,E1 -11024.031,E2 -11024.031} C_VEL
LIN {X 0,Y 406.378,Z 246.098,A -85,B 0,C 180,E1 -11025.203,E2 -11025.203} C_VEL
LIN {X 0,Y 410.902,Z 268.097,A -85,B 0,C 180,E1 -11025.859,E2 -11025.859} C_VEL
LIN {X 0,Y 409.508,Z 354.11,A -85,B 0,C 180,E1 -11027.424,E2 -11027.424} C_VEL
LIN {X 0,Y 409.094,Z 367.824,A -85,B 0,C 180,E1 -11027.892,E2 -11027.892} C_VEL
LIN {X 0,Y 408.502,Z 380.265,A -85,B 0,C 180,E1 -11028.52,E2 -11028.52} C_VEL
LIN {X 0,Y 407.806,Z 391.873,A -85,B 0,C 180,E1 -11029.313,E2 -11029.313} C_VEL
LIN {X 0,Y 407.007,Z 403.042,A -85,B 0,C 180,E1 -11030.29,E2 -11030.29} C_VEL
LIN {X 0,Y 406.131,Z 413.766,A -85,B 0,C 180,E1 -11031.467,E2 -11031.467} C_VEL
LIN {X 0,Y 405.386,Z 422.417,A -85,B 0,C 180,E1 -11032.643,E2 -11032.643} C_VEL
LIN {X 0,Y 404.664,Z 431.019,A -85,B 0,C 180,E1 -11034.081,E2 -11034.081} C_VEL
LIN {X 0,Y 404.027,Z 438.254,A -85,B 0,C 180,E1 -11035.575,E2 -11035.575} C_VEL
LIN {X 0,Y 403.617,Z 443.818,A -85,B 0,C 180,E1 -11037.006,E2 -11037.006} C_VEL
LIN {X 0,Y 403.302,Z 448.812,A -85,B 0,C 180,E1 -11038.637,E2 -11038.637} C_VEL
LIN {X 0,Y 403.057,Z 452.391,A -85,B 0,C 180,E1 -11040.202,E2 -11040.202} C_VEL
LIN {X 0,Y 402.802,Z 455.042,A -85,B 0,C 180,E1 -11041.895,E2 -11041.895} C_VEL
LIN {X 0,Y 402.711,Z 456.138,A -85,B 0,C 180,E1 -11043.016,E2 -11043.016} C_VEL
LIN {X 0,Y 402.646,Z 456.767,A -85,B 0,C 180,E1 -11044.128,E2 -11044.128} C_VEL
LIN {X 0,Y 402.624,Z 456.862,A -85,B 0,C 180,E1 -11045.233,E2 -11045.233} C_VEL
LIN {X 0,Y 402.637,Z 456.498,A -85,B 0,C 180,E1 -11046.33,E2 -11046.33} C_VEL
LIN {X 0,Y 402.715,Z 455.412,A -85,B 0,C 180,E1 -11047.659,E2 -11047.659} C_VEL
LIN {X 0,Y 402.975,Z 452.562,A -85,B 0,C 180,E1 -11049.586,E2 -11049.586} C_VEL
LIN {X 0,Y 403.23,Z 448.961,A -85,B 0,C 180,E1 -11051.189,E2 -11051.189} C_VEL
LIN {X 0,Y 403.48,Z 444.189,A -85,B 0,C 180,E1 -11052.776,E2 -11052.776} C_VEL
LIN {X 0,Y 403.933,Z 438.046,A -85,B 0,C 180,E1 -11054.355,E2 -11054.355} C_VEL
LIN {X 0,Y 404.519,Z 430.364,A -85,B 0,C 180,E1 -11055.923,E2 -11055.923} C_VEL
LIN {X 0,Y 405.172,Z 422.497,A -85,B 0,C 180,E1 -11057.223,E2 -11057.223} C_VEL
LIN {X 0,Y 405.902,Z 412.931,A -85,B 0,C 180,E1 -11058.515,E2 -11058.515} C_VEL
LIN {X 0,Y 406.726,Z 401.807,A -85,B 0,C 180,E1 -11059.71,E2 -11059.71} C_VEL
LIN {X 0,Y 407.593,Z 390.183,A -85,B 0,C 180,E1 -11060.697,E2 -11060.697} C_VEL
LIN {X 0,Y 408.196,Z 378.557,A -85,B 0,C 180,E1 -11061.46,E2 -11061.46} C_VEL
LIN {X 0,Y 408.692,Z 365.458,A -85,B 0,C 180,E1 -11062.093,E2 -11062.093} C_VEL
LIN {X 0,Y 409.101,Z 352.576,A -85,B 0,C 180,E1 -11062.504,E2 -11062.504} C_VEL
LIN {X 0,Y 409.307,Z 339.901,A -85,B 0,C 180,E1 -11062.746,E2 -11062.746} C_VEL
LIN {X 0,Y 408.802,Z 334.091,A -85,B 0,C 180,E1 -11062.875,E2 -11062.875} C_VEL
LIN {X 0,Y 403.587,Z 315.38,A -85,B 0,C 180,E1 -11063.45,E2 -11063.45} C_VEL
LIN {X 0,Y 402.955,Z 309.571,A -85,B 0,C 180,E1 -11063.587,E2 -11063.587} C_VEL
LIN {X 0,Y 403.443,Z 267.734,A -85,B 0,C 180,E1 -11064.352,E2 -11064.352} C_VEL
LIN {X 0,Y 399.173,Z 246.061,A -85,B 0,C 180,E1 -11064.981,E2 -11064.981} C_VEL
LIN {X 0,Y 399.183,Z 240.889,A -85,B 0,C 180,E1 -11066.214,E2 -11066.214} C_VEL
LIN {X 0,Y 397.547,Z 230.891,A -85,B 0,C 180,E1 -11068.734,E2 -11068.734} C_VEL
LIN {X 0,Y 397.365,Z 229.988,A -85,B 0,C 180,E1 -11068.986,E2 -11068.986} C_VEL
LIN {X 0,Y 397.444,Z 229.977,A -85,B 0,C 180,E1 -11072.027,E2 -11072.027} C_VEL
LIN {X 0,Y 397.332,Z 229.991,A -85,B 0,C 180,E1 -11076.092,E2 -11076.092} C_VEL
LIN {X 0,Y 397.238,Z 230.001,A -85,B 0,C 180,E1 -11079.162,E2 -11079.162} C_VEL
LIN {X 0,Y 397.221,Z 230.004,A -85,B 0,C 180,E1 -11082.258,E2 -11082.258} C_VEL
LIN {X 0,Y 397.178,Z 230.01,A -85,B 0,C 180,E1 -11085.392,E2 -11085.392} C_VEL
LIN {X 0,Y 397.162,Z 230.01,A -85,B 0,C 180,E1 -11088.573,E2 -11088.573} C_VEL
LIN {X 0,Y 397.099,Z 230.023,A -85,B 0,C 180,E1 -11091.818,E2 -11091.818} C_VEL
LIN {X 0,Y 397.125,Z 230.015,A -85,B 0,C 180,E1 -11095.133,E2 -11095.133} C_VEL
LIN {X 0,Y 397.08,Z 230.021,A -85,B 0,C 180,E1 -11098.547,E2 -11098.547} C_VEL
LIN {X 0,Y 397.083,Z 230.025,A -85,B 0,C 180,E1 -11101.836,E2 -11101.836} C_VEL
LIN {X 0,Y 397.126,Z 230.016,A -85,B 0,C 180,E1 -11104.493,E2 -11104.493} C_VEL
LIN {X 0,Y 397.098,Z 230.021,A -85,B 0,C 180,E1 -11108.275,E2 -11108.275} C_VEL
LIN {X 0,Y 397.062,Z 230.023,A -85,B 0,C 180,E1 -11110.911,E2 -11110.911} C_VEL
LIN {X 0,Y 397.099,Z 230.022,A -85,B 0,C 180,E1 -11113.648,E2 -11113.648} C_VEL
LIN {X 0,Y 397.101,Z 230.02,A -85,B 0,C 180,E1 -11116.521,E2 -11116.521} C_VEL
LIN {X 0,Y 397.112,Z 230.019,A -85,B 0,C 180,E1 -11120.422,E2 -11120.422} C_VEL
LIN {X 0,Y 397.107,Z 230.02,A -85,B 0,C 180,E1 -11124.265,E2 -11124.265} C_VEL
LIN {X 0,Y 397.113,Z 230.017,A -85,B 0,C 180,E1 -11126.727,E2 -11126.727} C_VEL
LIN {X 0,Y 397.123,Z 230.019,A -85,B 0,C 180,E1 -11130.295,E2 -11130.295} C_VEL
LIN {X 0,Y 397.192,Z 230.008,A -85,B 0,C 180,E1 -11132.609,E2 -11132.609} C_VEL
LIN {X 0,Y 397.131,Z 230.018,A -85,B 0,C 180,E1 -11135.981,E2 -11135.981} C_VEL
LIN {X 0,Y 397.136,Z 230.017,A -85,B 0,C 180,E1 -11139.704,E2 -11139.704} C_VEL
LIN {X 0,Y 397.179,Z 230.009,A -85,B 0,C 180,E1 -11142.845,E2 -11142.845} C_VEL
LIN {X 0,Y 397.226,Z 230.004,A -85,B 0,C 180,E1 -11146.702,E2 -11146.702} C_VEL
LIN {X 0,Y 397.215,Z 230.008,A -85,B 0,C 180,E1 -11149.809,E2 -11149.809} C_VEL
LIN {X 0,Y 397.362,Z 229.986,A -85,B 0,C 180,E1 -11152.888,E2 -11152.888} C_VEL
LIN {X 0,Y 397.253,Z 230,A -85,B 0,C 180,E1 -11154.925,E2 -11154.925} C_VEL
LIN {X 0,Y 397.449,Z 229.978,A -85,B 0,C 180,E1 -11157.973,E2 -11157.973} C_VEL
LIN {X 0,Y 397.576,Z 229.962,A -85,B 0,C 180,E1 -11160,E2 -11160} C_VEL
LIN {X 0,Y 397.379,Z 229.984,A -85,B 0,C 180,E1 -11163.041,E2 -11163.041} C_VEL
LIN {X 0,Y 397.361,Z 229.986,A -85,B 0,C 180,E1 -11167.112,E2 -11167.112} C_VEL
LIN {X 0,Y 397.215,Z 230.007,A -85,B 0,C 180,E1 -11170.191,E2 -11170.191} C_VEL
LIN {X 0,Y 397.224,Z 230.003,A -85,B 0,C 180,E1 -11173.321,E2 -11173.321} C_VEL
LIN {X 0,Y 397.179,Z 230.008,A -85,B 0,C 180,E1 -11177.155,E2 -11177.155} C_VEL
LIN {X 0,Y 397.1,Z 230.02,A -85,B 0,C 180,E1 -11180.73,E2 -11180.73} C_VEL
LIN {X 0,Y 397.131,Z 230.017,A -85,B 0,C 180,E1 -11184.018,E2 -11184.018} C_VEL
LIN {X 0,Y 397.192,Z 230.007,A -85,B 0,C 180,E1 -11187.39,E2 -11187.39} C_VEL
LIN {X 0,Y 397.076,Z 230.022,A -85,B 0,C 180,E1 -11190.883,E2 -11190.883} C_VEL
LIN {X 0,Y 397.124,Z 230.02,A -85,B 0,C 180,E1 -11194.494,E2 -11194.494} C_VEL
LIN {X 0,Y 397.101,Z 230.022,A -85,B 0,C 180,E1 -11198.275,E2 -11198.275} C_VEL
LIN {X 0,Y 397.087,Z 230.021,A -85,B 0,C 180,E1 -11200.909,E2 -11200.909} C_VEL
LIN {X 0,Y 397.099,Z 230.018,A -85,B 0,C 180,E1 -11203.649,E2 -11203.649} C_VEL
LIN {X 0,Y 397.101,Z 230.023,A -85,B 0,C 180,E1 -11206.521,E2 -11206.521} C_VEL
LIN {X 0,Y 397.113,Z 230.021,A -85,B 0,C 180,E1 -11210.423,E2 -11210.423} C_VEL
LIN {X 0,Y 397.107,Z 230.02,A -85,B 0,C 180,E1 -11214.266,E2 -11214.266} C_VEL
LIN {X 0,Y 397.114,Z 230.022,A -85,B 0,C 180,E1 -11216.728,E2 -11216.728} C_VEL
LIN {X 0,Y 397.125,Z 230.019,A -85,B 0,C 180,E1 -11220.296,E2 -11220.296} C_VEL
LIN {X 0,Y 397.223,Z 230.181,A -85,B 0,C 180,E1 -11221.994,E2 -11221.994} C_VEL
LIN {X 0,Y 399.75,Z 243.217,A -85,B 0,C 180,E1 -11225.043,E2 -11225.043} C_VEL
LIN {X 0,Y 400.329,Z 247.044,A -85,B 0,C 180,E1 -11225.908,E2 -11225.908} C_VEL
LIN {X 0,Y 399.265,Z 261.194,A -85,B 0,C 180,E1 -11228.896,E2 -11228.896} C_VEL
LIN {X 0,Y 398.865,Z 266.655,A -85,B 0,C 180,E1 -11230.039,E2 -11230.039} C_VEL
LIN {X 0,Y 403.295,Z 294.868,A -85,B 0,C 180,E1 -11230.789,E2 -11230.789} C_VEL
LIN {X 0,Y 402.202,Z 374.763,A -85,B 0,C 180,E1 -11232.26,E2 -11232.26} C_VEL
LIN {X 0,Y 401.666,Z 387.99,A -85,B 0,C 180,E1 -11232.696,E2 -11232.696} C_VEL
LIN {X 0,Y 400.976,Z 400.721,A -85,B 0,C 180,E1 -11233.321,E2 -11233.321} C_VEL
LIN {X 0,Y 400.229,Z 412.048,A -85,B 0,C 180,E1 -11234.076,E2 -11234.076} C_VEL
LIN {X 0,Y 399.342,Z 424.132,A -85,B 0,C 180,E1 -11235.124,E2 -11235.124} C_VEL
LIN {X 0,Y 398.573,Z 434.651,A -85,B 0,C 180,E1 -11236.276,E2 -11236.276} C_VEL
LIN {X 0,Y 397.835,Z 443.731,A -85,B 0,C 180,E1 -11237.502,E2 -11237.502} C_VEL
LIN {X 0,Y 396.996,Z 452.848,A -85,B 0,C 180,E1 -11239.03,E2 -11239.03} C_VEL
LIN {X 0,Y 396.487,Z 460.199,A -85,B 0,C 180,E1 -11240.563,E2 -11240.563} C_VEL
LIN {X 0,Y 396.185,Z 465.177,A -85,B 0,C 180,E1 -11241.842,E2 -11241.842} C_VEL
LIN {X 0,Y 395.937,Z 470.007,A -85,B 0,C 180,E1 -11243.375,E2 -11243.375} C_VEL
LIN {X 0,Y 395.843,Z 473.706,A -85,B 0,C 180,E1 -11244.907,E2 -11244.907} C_VEL
LIN {X 0,Y 395.774,Z 475.615,A -85,B 0,C 180,E1 -11245.927,E2 -11245.927} C_VEL
LIN {X 0,Y 395.728,Z 477.073,A -85,B 0,C 180,E1 -11246.946,E2 -11246.946} C_VEL
LIN {X 0,Y 395.763,Z 478.101,A -85,B 0,C 180,E1 -11247.965,E2 -11247.965} C_VEL
LIN {X 0,Y 395.791,Z 478.736,A -85,B 0,C 180,E1 -11248.983,E2 -11248.983} C_VEL
LIN {X 0,Y 395.779,Z 478.982,A -85,B 0,C 180,E1 -11250,E2 -11250} C_VEL
LIN {X 0,Y 395.791,Z 478.808,A -85,B 0,C 180,E1 -11251.018,E2 -11251.018} C_VEL
LIN {X 0,Y 395.762,Z 478.216,A -85,B 0,C 180,E1 -11252.036,E2 -11252.036} C_VEL
LIN {X 0,Y 395.774,Z 475.855,A -85,B 0,C 180,E1 -11254.073,E2 -11254.073} C_VEL
LIN {X 0,Y 395.826,Z 472.499,A -85,B 0,C 180,E1 -11255.805,E2 -11255.805} C_VEL
LIN {X 0,Y 396.073,Z 467.426,A -85,B 0,C 180,E1 -11257.648,E2 -11257.648} C_VEL
LIN {X 0,Y 396.51,Z 460.916,A -85,B 0,C 180,E1 -11259.437,E2 -11259.437} C_VEL
LIN {X 0,Y 397.038,Z 453.784,A -85,B 0,C 180,E1 -11260.97,E2 -11260.97} C_VEL
LIN {X 0,Y 397.896,Z 444.904,A -85,B 0,C 180,E1 -11262.496,E2 -11262.496} C_VEL
LIN {X 0,Y 398.766,Z 434.92,A -85,B 0,C 180,E1 -11263.881,E2 -11263.881} C_VEL
LIN {X 0,Y 399.534,Z 424.753,A -85,B 0,C 180,E1 -11265.012,E2 -11265.012} C_VEL
LIN {X 0,Y 400.486,Z 413.071,A -85,B 0,C 180,E1 -11266.045,E2 -11266.045} C_VEL
LIN {X 0,Y 401.345,Z 401.187,A -85,B 0,C 180,E1 -11266.86,E2 -11266.86} C_VEL
LIN {X 0,Y 402.161,Z 388.043,A -85,B 0,C 180,E1 -11267.512,E2 -11267.512} C_VEL
LIN {X 0,Y 402.687,Z 375.073,A -85,B 0,C 180,E1 -11267.948,E2 -11267.948} C_VEL
LIN {X 0,Y 403.885,Z 295.043,A -85,B 0,C 180,E1 -11269.434,E2 -11269.434} C_VEL
LIN {X 0,Y 400.103,Z 271.607,A -85,B 0,C 180,E1 -11270.088,E2 -11270.088} C_VEL
LIN {X 0,Y 399.09,Z 265.897,A -85,B 0,C 180,E1 -11270.284,E2 -11270.284} C_VEL
LIN {X 0,Y 400.311,Z 248.905,A -85,B 0,C 180,E1 -11273.816,E2 -11273.816} C_VEL
LIN {X 0,Y 400.165,Z 244.877,A -85,B 0,C 180,E1 -11274.691,E2 -11274.691} C_VEL
LIN {X 0,Y 397.464,Z 231.284,A -85,B 0,C 180,E1 -11277.858,E2 -11277.858} C_VEL
LIN {X 0,Y 397.179,Z 230.013,A -85,B 0,C 180,E1 -11278.225,E2 -11278.225} C_VEL
LIN {X 0,Y 397.08,Z 230.026,A -85,B 0,C 180,E1 -11282.071,E2 -11282.071} C_VEL
LIN {X 0,Y 397.12,Z 230.02,A -85,B 0,C 180,E1 -11285.503,E2 -11285.503} C_VEL
LIN {X 0,Y 397.128,Z 230.017,A -85,B 0,C 180,E1 -11288.861,E2 -11288.861} C_VEL
LIN {X 0,Y 397.071,Z 230.021,A -85,B 0,C 180,E1 -11292.267,E2 -11292.267} C_VEL
LIN {X 0,Y 397.089,Z 230.022,A -85,B 0,C 180,E1 -11295.068,E2 -11295.068} C_VEL
LIN {X 0,Y 397.066,Z 230.019,A -85,B 0,C 180,E1 -11298.021,E2 -11298.021} C_VEL
LIN {X 0,Y 397.128,Z 230.015,A -85,B 0,C 180,E1 -11301.139,E2 -11301.139} C_VEL
LIN {X 0,Y 397.119,Z 230.014,A -85,B 0,C 180,E1 -11304.496,E2 -11304.496} C_VEL
LIN {X 0,Y 397.078,Z 230.017,A -85,B 0,C 180,E1 -11307.928,E2 -11307.928} C_VEL
LIN {X 0,Y 397.122,Z 230.014,A -85,B 0,C 180,E1 -11311.456,E2 -11311.456} C_VEL
LIN {X 0,Y 397.152,Z 230.012,A -85,B 0,C 180,E1 -11314.488,E2 -11314.488} C_VEL
LIN {X 0,Y 397.108,Z 230.015,A -85,B 0,C 180,E1 -11317.086,E2 -11317.086} C_VEL
LIN {X 0,Y 397.147,Z 230.012,A -85,B 0,C 180,E1 -11320.353,E2 -11320.353} C_VEL
LIN {X 0,Y 397.166,Z 230.01,A -85,B 0,C 180,E1 -11323.553,E2 -11323.553} C_VEL
LIN {X 0,Y 397.228,Z 229.997,A -85,B 0,C 180,E1 -11326.703,E2 -11326.703} C_VEL
LIN {X 0,Y 397.217,Z 229.998,A -85,B 0,C 180,E1 -11329.809,E2 -11329.809} C_VEL
LIN {X 0,Y 397.349,Z 229.992,A -85,B 0,C 180,E1 -11332.888,E2 -11332.888} C_VEL
LIN {X 0,Y 397.253,Z 229.996,A -85,B 0,C 180,E1 -11334.925,E2 -11334.925} C_VEL
LIN {X 0,Y 397.451,Z 229.974,A -85,B 0,C 180,E1 -11337.973,E2 -11337.973} C_VEL
LIN {X 0,Y 397.578,Z 229.952,A -85,B 0,C 180,E1 -11340,E2 -11340} C_VEL
LIN {X 0,Y 397.378,Z 229.982,A -85,B 0,C 180,E1 -11343.042,E2 -11343.042} C_VEL
LIN {X 0,Y 397.362,Z 229.984,A -85,B 0,C 180,E1 -11347.112,E2 -11347.112} C_VEL
LIN {X 0,Y 397.217,Z 230.005,A -85,B 0,C 180,E1 -11350.191,E2 -11350.191} C_VEL
LIN {X 0,Y 397.226,Z 230.004,A -85,B 0,C 180,E1 -11353.321,E2 -11353.321} C_VEL
LIN {X 0,Y 397.182,Z 230.009,A -85,B 0,C 180,E1 -11357.155,E2 -11357.155} C_VEL
LIN {X 0,Y 397.102,Z 230.02,A -85,B 0,C 180,E1 -11360.73,E2 -11360.73} C_VEL
LIN {X 0,Y 397.123,Z 230.015,A -85,B 0,C 180,E1 -11364.019,E2 -11364.019} C_VEL
LIN {X 0,Y 397.115,Z 230.017,A -85,B 0,C 180,E1 -11367.763,E2 -11367.763} C_VEL
LIN {X 0,Y 397.078,Z 230.024,A -85,B 0,C 180,E1 -11370.883,E2 -11370.883} C_VEL
LIN {X 0,Y 397.124,Z 230.02,A -85,B 0,C 180,E1 -11374.494,E2 -11374.494} C_VEL
LIN {X 0,Y 397.09,Z 230.027,A -85,B 0,C 180,E1 -11378.277,E2 -11378.277} C_VEL
LIN {X 0,Y 397.092,Z 230.024,A -85,B 0,C 180,E1 -11380.993,E2 -11380.993} C_VEL
LIN {X 0,Y 399.108,Z 239.801,A -85,B 0,C 180,E1 -11383.375,E2 -11383.375} C_VEL
LIN {X 0,Y 399.608,Z 244.003,A -85,B 0,C 180,E1 -11384.358,E2 -11384.358} C_VEL
LIN {X 0,Y 399.516,Z 246.301,A -85,B 0,C 180,E1 -11384.825,E2 -11384.825} C_VEL
LIN {X 0,Y 404.17,Z 268.411,A -85,B 0,C 180,E1 -11385.511,E2 -11385.511} C_VEL
LIN {X 0,Y 402.847,Z 353.517,A -85,B 0,C 180,E1 -11387.084,E2 -11387.084} C_VEL
LIN {X 0,Y 402.394,Z 366.948,A -85,B 0,C 180,E1 -11387.534,E2 -11387.534} C_VEL
LIN {X 0,Y 401.78,Z 379.713,A -85,B 0,C 180,E1 -11388.173,E2 -11388.173} C_VEL
LIN {X 0,Y 401.031,Z 391.607,A -85,B 0,C 180,E1 -11388.986,E2 -11388.986} C_VEL
LIN {X 0,Y 400.211,Z 402.795,A -85,B 0,C 180,E1 -11389.973,E2 -11389.973} C_VEL
LIN {X 0,Y 399.287,Z 413.607,A -85,B 0,C 180,E1 -11391.167,E2 -11391.167} C_VEL
LIN {X 0,Y 398.381,Z 423.514,A -85,B 0,C 180,E1 -11392.549,E2 -11392.549} C_VEL
LIN {X 0,Y 397.655,Z 431.956,A -85,B 0,C 180,E1 -11394.01,E2 -11394.01} C_VEL
LIN {X 0,Y 396.991,Z 438.901,A -85,B 0,C 180,E1 -11395.493,E2 -11395.493} C_VEL
LIN {X 0,Y 396.484,Z 445.414,A -85,B 0,C 180,E1 -11397.273,E2 -11397.273} C_VEL
LIN {X 0,Y 396.149,Z 450.299,A -85,B 0,C 180,E1 -11399.037,E2 -11399.037} C_VEL
LIN {X 0,Y 395.942,Z 453.164,A -85,B 0,C 180,E1 -11400.431,E2 -11400.431} C_VEL
LIN {X 0,Y 395.649,Z 455.963,A -85,B 0,C 180,E1 -11402.494,E2 -11402.494} C_VEL
LIN {X 0,Y 395.562,Z 456.751,A -85,B 0,C 180,E1 -11403.629,E2 -11403.629} C_VEL
LIN {X 0,Y 395.532,Z 457.096,A -85,B 0,C 180,E1 -11404.985,E2 -11404.985} C_VEL
LIN {X 0,Y 395.587,Z 456.254,A -85,B 0,C 180,E1 -11406.992,E2 -11406.992} C_VEL
LIN {X 0,Y 395.69,Z 455.153,A -85,B 0,C 180,E1 -11408.1,E2 -11408.1} C_VEL
LIN {X 0,Y 395.82,Z 453.555,A -85,B 0,C 180,E1 -11409.2,E2 -11409.2} C_VEL
LIN {X 0,Y 396.091,Z 450.247,A -85,B 0,C 180,E1 -11410.837,E2 -11410.837} C_VEL
LIN {X 0,Y 396.33,Z 445.8,A -85,B 0,C 180,E1 -11412.455,E2 -11412.455} C_VEL
LIN {X 0,Y 396.731,Z 440.071,A -85,B 0,C 180,E1 -11414.063,E2 -11414.063} C_VEL
LIN {X 0,Y 397.359,Z 432.864,A -85,B 0,C 180,E1 -11415.664,E2 -11415.664} C_VEL
LIN {X 0,Y 397.97,Z 425.474,A -85,B 0,C 180,E1 -11416.988,E2 -11416.988} C_VEL
LIN {X 0,Y 398.788,Z 415.466,A -85,B 0,C 180,E1 -11418.436,E2 -11418.436} C_VEL
LIN {X 0,Y 399.609,Z 405.351,A -85,B 0,C 180,E1 -11419.615,E2 -11419.615} C_VEL
LIN {X 0,Y 400.318,Z 395.693,A -85,B 0,C 180,E1 -11420.527,E2 -11420.527} C_VEL
LIN {X 0,Y 401.103,Z 383.515,A -85,B 0,C 180,E1 -11421.435,E2 -11421.435} C_VEL
LIN {X 0,Y 401.681,Z 370.861,A -85,B 0,C 180,E1 -11422.143,E2 -11422.143} C_VEL
LIN {X 0,Y 402.187,Z 358.52,A -85,B 0,C 180,E1 -11422.627,E2 -11422.627} C_VEL
LIN {X 0,Y 402.452,Z 345.002,A -85,B 0,C 180,E1 -11422.947,E2 -11422.947} C_VEL
LIN {X 0,Y 402.955,Z 309.571,A -85,B 0,C 180,E1 -11423.587,E2 -11423.587} C_VEL
LIN {X 0,Y 402.338,Z 303.766,A -85,B 0,C 180,E1 -11423.724,E2 -11423.724} C_VEL
LIN {X 0,Y 397.215,Z 285.059,A -85,B 0,C 180,E1 -11424.319,E2 -11424.319} C_VEL
LIN {X 0,Y 396.685,Z 279.253,A -85,B 0,C 180,E1 -11424.456,E2 -11424.456} C_VEL
LIN {X 0,Y 396.688,Z 268.617,A -85,B 0,C 180,E1 -11424.661,E2 -11424.661} C_VEL
LIN {X 0,Y 392.294,Z 246.168,A -85,B 0,C 180,E1 -11425.344,E2 -11425.344} C_VEL
LIN {X 0,Y 392.161,Z 241.834,A -85,B 0,C 180,E1 -11426.404,E2 -11426.404} C_VEL
LIN {X 0,Y 390.92,Z 233.796,A -85,B 0,C 180,E1 -11428.455,E2 -11428.455} C_VEL
LIN {X 0,Y 390.333,Z 230.861,A -85,B 0,C 180,E1 -11429.226,E2 -11429.226} C_VEL
LIN {X 0,Y 390.411,Z 230.853,A -85,B 0,C 180,E1 -11432.063,E2 -11432.063} C_VEL
LIN {X 0,Y 390.286,Z 230.868,A -85,B 0,C 180,E1 -11436.202,E2 -11436.202} C_VEL
LIN {X 0,Y 390.195,Z 230.879,A -85,B 0,C 180,E1 -11439.329,E2 -11439.329} C_VEL
LIN {X 0,Y 390.173,Z 230.881,A -85,B 0,C 180,E1 -11442.483,E2 -11442.483} C_VEL
LIN {X 0,Y 390.139,Z 230.89,A -85,B 0,C 180,E1 -11445.677,E2 -11445.677} C_VEL
LIN {X 0,Y 390.106,Z 230.889,A -85,B 0,C 180,E1 -11448.922,E2 -11448.922} C_VEL
LIN {X 0,Y 390.041,Z 230.899,A -85,B 0,C 180,E1 -11452.234,E2 -11452.234} C_VEL
LIN {X 0,Y 390.085,Z 230.897,A -85,B 0,C 180,E1 -11455.732,E2 -11455.732} C_VEL
LIN {X 0,Y 390.034,Z 230.898,A -85,B 0,C 180,E1 -11459.111,E2 -11459.111} C_VEL
LIN {X 0,Y 390.044,Z 230.897,A -85,B 0,C 180,E1 -11462.721,E2 -11462.721} C_VEL
LIN {X 0,Y 390.056,Z 230.9,A -85,B 0,C 180,E1 -11465.825,E2 -11465.825} C_VEL
LIN {X 0,Y 390.061,Z 230.895,A -85,B 0,C 180,E1 -11469.216,E2 -11469.216} C_VEL
LIN {X 0,Y 390.038,Z 230.9,A -85,B 0,C 180,E1 -11472.373,E2 -11472.373} C_VEL
LIN {X 0,Y 390.043,Z 230.898,A -85,B 0,C 180,E1 -11475.354,E2 -11475.354} C_VEL
LIN {X 0,Y 390.03,Z 230.902,A -85,B 0,C 180,E1 -11478.186,E2 -11478.186} C_VEL
LIN {X 0,Y 390.087,Z 230.892,A -85,B 0,C 180,E1 -11480.907,E2 -11480.907} C_VEL
LIN {X 0,Y 390.084,Z 230.892,A -85,B 0,C 180,E1 -11484.793,E2 -11484.793} C_VEL
LIN {X 0,Y 390.022,Z 230.902,A -85,B 0,C 180,E1 -11488.495,E2 -11488.495} C_VEL
LIN {X 0,Y 390.115,Z 230.892,A -85,B 0,C 180,E1 -11492.07,E2 -11492.07} C_VEL
LIN {X 0,Y 390.078,Z 230.894,A -85,B 0,C 180,E1 -11495.519,E2 -11495.519} C_VEL
LIN {X 0,Y 390.053,Z 230.896,A -85,B 0,C 180,E1 -11498.877,E2 -11498.877} C_VEL
LIN {X 0,Y 390.126,Z 230.891,A -85,B 0,C 180,E1 -11502.166,E2 -11502.166} C_VEL
LIN {X 0,Y 390.141,Z 230.886,A -85,B 0,C 180,E1 -11505.392,E2 -11505.392} C_VEL
LIN {X 0,Y 390.146,Z 230.887,A -85,B 0,C 180,E1 -11508.571,E2 -11508.571} C_VEL
LIN {X 0,Y 390.341,Z 230.864,A -85,B 0,C 180,E1 -11511.993,E2 -11511.993} C_VEL
LIN {X 0,Y 390.225,Z 230.875,A -85,B 0,C 180,E1 -11514.833,E2 -11514.833} C_VEL
LIN {X 0,Y 390.418,Z 230.854,A -85,B 0,C 180,E1 -11517.937,E2 -11517.937} C_VEL
LIN {X 0,Y 390.545,Z 230.838,A -85,B 0,C 180,E1 -11520,E2 -11520} C_VEL
LIN {X 0,Y 390.313,Z 230.864,A -85,B 0,C 180,E1 -11523.096,E2 -11523.096} C_VEL
LIN {X 0,Y 390.328,Z 230.865,A -85,B 0,C 180,E1 -11526.202,E2 -11526.202} C_VEL
LIN {X 0,Y 390.312,Z 230.868,A -85,B 0,C 180,E1 -11528.282,E2 -11528.282} C_VEL
LIN {X 0,Y 390.168,Z 230.886,A -85,B 0,C 180,E1 -11532.483,E2 -11532.483} C_VEL
LIN {X 0,Y 390.136,Z 230.887,A -85,B 0,C 180,E1 -11535.677,E2 -11535.677} C_VEL
LIN {X 0,Y 390.103,Z 230.89,A -85,B 0,C 180,E1 -11538.922,E2 -11538.922} C_VEL
LIN {X 0,Y 390.038,Z 230.902,A -85,B 0,C 180,E1 -11542.234,E2 -11542.234} C_VEL
LIN {X 0,Y 390.117,Z 230.889,A -85,B 0,C 180,E1 -11545.744,E2 -11545.744} C_VEL
LIN {X 0,Y 390.056,Z 230.895,A -85,B 0,C 180,E1 -11549.11,E2 -11549.11} C_VEL
LIN {X 0,Y 390.041,Z 230.9,A -85,B 0,C 180,E1 -11552.722,E2 -11552.722} C_VEL
LIN {X 0,Y 390.054,Z 230.897,A -85,B 0,C 180,E1 -11555.826,E2 -11555.826} C_VEL
LIN {X 0,Y 390.067,Z 230.894,A -85,B 0,C 180,E1 -11559.219,E2 -11559.219} C_VEL
LIN {X 0,Y 390.041,Z 230.902,A -85,B 0,C 180,E1 -11562.375,E2 -11562.375} C_VEL
LIN {X 0,Y 390.043,Z 230.896,A -85,B 0,C 180,E1 -11565.355,E2 -11565.355} C_VEL
LIN {X 0,Y 390.03,Z 230.901,A -85,B 0,C 180,E1 -11568.187,E2 -11568.187} C_VEL
LIN {X 0,Y 390.089,Z 230.892,A -85,B 0,C 180,E1 -11570.908,E2 -11570.908} C_VEL
LIN {X 0,Y 390.084,Z 230.894,A -85,B 0,C 180,E1 -11574.794,E2 -11574.794} C_VEL
LIN {X 0,Y 390.024,Z 230.905,A -85,B 0,C 180,E1 -11578.496,E2 -11578.496} C_VEL
LIN {X 0,Y 390.149,Z 230.974,A -85,B 0,C 180,E1 -11581.694,E2 -11581.694} C_VEL
LIN {X 0,Y 392.51,Z 242.912,A -85,B 0,C 180,E1 -11584.55,E2 -11584.55} C_VEL
LIN {X 0,Y 393.359,Z 248.03,A -85,B 0,C 180,E1 -11585.737,E2 -11585.737} C_VEL
LIN {X 0,Y 392.305,Z 261.72,A -85,B 0,C 180,E1 -11588.68,E2 -11588.68} C_VEL
LIN {X 0,Y 391.975,Z 266.508,A -85,B 0,C 180,E1 -11589.699,E2 -11589.699} C_VEL
LIN {X 0,Y 396.536,Z 295.349,A -85,B 0,C 180,E1 -11590.482,E2 -11590.482} C_VEL
LIN {X 0,Y 395.392,Z 374.961,A -85,B 0,C 180,E1 -11591.978,E2 -11591.978} C_VEL
LIN {X 0,Y 394.837,Z 388.057,A -85,B 0,C 180,E1 -11592.42,E2 -11592.42} C_VEL
LIN {X 0,Y 394.148,Z 400.153,A -85,B 0,C 180,E1 -11593.024,E2 -11593.024} C_VEL
LIN {X 0,Y 393.376,Z 411.582,A -85,B 0,C 180,E1 -11593.791,E2 -11593.791} C_VEL
LIN {X 0,Y 392.482,Z 423.335,A -85,B 0,C 180,E1 -11594.818,E2 -11594.818} C_VEL
LIN {X 0,Y 391.731,Z 433.413,A -85,B 0,C 180,E1 -11595.924,E2 -11595.924} C_VEL
LIN {X 0,Y 390.884,Z 443.406,A -85,B 0,C 180,E1 -11597.276,E2 -11597.276} C_VEL
LIN {X 0,Y 389.998,Z 452.552,A -85,B 0,C 180,E1 -11598.83,E2 -11598.83} C_VEL
LIN {X 0,Y 389.462,Z 459.925,A -85,B 0,C 180,E1 -11600.391,E2 -11600.391} C_VEL
LIN {X 0,Y 389.128,Z 464.92,A -85,B 0,C 180,E1 -11601.693,E2 -11601.693} C_VEL
LIN {X 0,Y 388.852,Z 469.763,A -85,B 0,C 180,E1 -11603.254,E2 -11603.254} C_VEL
LIN {X 0,Y 388.739,Z 473.477,A -85,B 0,C 180,E1 -11604.814,E2 -11604.814} C_VEL
LIN {X 0,Y 388.699,Z 475.393,A -85,B 0,C 180,E1 -11605.853,E2 -11605.853} C_VEL
LIN {X 0,Y 388.635,Z 476.86,A -85,B 0,C 180,E1 -11606.89,E2 -11606.89} C_VEL
LIN {X 0,Y 388.661,Z 477.892,A -85,B 0,C 180,E1 -11607.928,E2 -11607.928} C_VEL
LIN {X 0,Y 388.703,Z 478.533,A -85,B 0,C 180,E1 -11608.964,E2 -11608.964} C_VEL
LIN {X 0,Y 388.708,Z 478.783,A -85,B 0,C 180,E1 -11610,E2 -11610} C_VEL
LIN {X 0,Y 388.703,Z 478.618,A -85,B 0,C 180,E1 -11611.036,E2 -11611.036} C_VEL
LIN {X 0,Y 388.66,Z 478.03,A -85,B 0,C 180,E1 -11612.073,E2 -11612.073} C_VEL
LIN {X 0,Y 388.699,Z 475.679,A -85,B 0,C 180,E1 -11614.148,E2 -11614.148} C_VEL
LIN {X 0,Y 388.727,Z 472.681,A -85,B 0,C 180,E1 -11615.754,E2 -11615.754} C_VEL
LIN {X 0,Y 388.936,Z 468.846,A -85,B 0,C 180,E1 -11617.267,E2 -11617.267} C_VEL
LIN {X 0,Y 389.261,Z 463.782,A -85,B 0,C 180,E1 -11618.828,E2 -11618.828} C_VEL
LIN {X 0,Y 389.782,Z 457.428,A -85,B 0,C 180,E1 -11620.388,E2 -11620.388} C_VEL
LIN {X 0,Y 390.477,Z 449.476,A -85,B 0,C 180,E1 -11621.946,E2 -11621.946} C_VEL
LIN {X 0,Y 391.281,Z 441.386,A -85,B 0,C 180,E1 -11623.239,E2 -11623.239} C_VEL
LIN {X 0,Y 392.1,Z 431.33,A -85,B 0,C 180,E1 -11624.557,E2 -11624.557} C_VEL
LIN {X 0,Y 393.05,Z 420.515,A -85,B 0,C 180,E1 -11625.691,E2 -11625.691} C_VEL
LIN {X 0,Y 393.924,Z 409.738,A -85,B 0,C 180,E1 -11626.586,E2 -11626.586} C_VEL
LIN {X 0,Y 394.887,Z 396.772,A -85,B 0,C 180,E1 -11627.411,E2 -11627.411} C_VEL
LIN {X 0,Y 395.585,Z 384.351,A -85,B 0,C 180,E1 -11627.98,E2 -11627.98} C_VEL
LIN {X 0,Y 396.086,Z 371.532,A -85,B 0,C 180,E1 -11628.358,E2 -11628.358} C_VEL
LIN {X 0,Y 397.082,Z 294.815,A -85,B 0,C 180,E1 -11629.802,E2 -11629.802} C_VEL
LIN {X 0,Y 392.844,Z 269.197,A -85,B 0,C 180,E1 -11630.545,E2 -11630.545} C_VEL
LIN {X 0,Y 392.196,Z 265.779,A -85,B 0,C 180,E1 -11630.661,E2 -11630.661} C_VEL
LIN {X 0,Y 393.406,Z 250.099,A -85,B 0,C 180,E1 -11633.98,E2 -11633.98} C_VEL
LIN {X 0,Y 393.242,Z 246.253,A -85,B 0,C 180,E1 -11634.833,E2 -11634.833} C_VEL
LIN {X 0,Y 390.702,Z 233.396,A -85,B 0,C 180,E1 -11637.885,E2 -11637.885} C_VEL
LIN {X 0,Y 390.129,Z 230.888,A -85,B 0,C 180,E1 -11638.532,E2 -11638.532} C_VEL
LIN {X 0,Y 390.033,Z 230.904,A -85,B 0,C 180,E1 -11642.124,E2 -11642.124} C_VEL
LIN {X 0,Y 390.085,Z 230.899,A -85,B 0,C 180,E1 -11645.207,E2 -11645.207} C_VEL
LIN {X 0,Y 390.069,Z 230.899,A -85,B 0,C 180,E1 -11649.218,E2 -11649.218} C_VEL
LIN {X 0,Y 390.044,Z 230.896,A -85,B 0,C 180,E1 -11652.374,E2 -11652.374} C_VEL
LIN {X 0,Y 390.046,Z 230.899,A -85,B 0,C 180,E1 -11655.354,E2 -11655.354} C_VEL
LIN {X 0,Y 390.031,Z 230.895,A -85,B 0,C 180,E1 -11658.187,E2 -11658.187} C_VEL
LIN {X 0,Y 390.088,Z 230.893,A -85,B 0,C 180,E1 -11660.907,E2 -11660.907} C_VEL
LIN {X 0,Y 390.085,Z 230.891,A -85,B 0,C 180,E1 -11664.793,E2 -11664.793} C_VEL
LIN {X 0,Y 390.023,Z 230.897,A -85,B 0,C 180,E1 -11668.496,E2 -11668.496} C_VEL
LIN {X 0,Y 390.117,Z 230.884,A -85,B 0,C 180,E1 -11672.07,E2 -11672.07} C_VEL
LIN {X 0,Y 390.08,Z 230.892,A -85,B 0,C 180,E1 -11675.519,E2 -11675.519} C_VEL
LIN {X 0,Y 390.055,Z 230.899,A -85,B 0,C 180,E1 -11678.878,E2 -11678.878} C_VEL
LIN {X 0,Y 390.127,Z 230.882,A -85,B 0,C 180,E1 -11682.167,E2 -11682.167} C_VEL
LIN {X 0,Y 390.144,Z 230.878,A -85,B 0,C 180,E1 -11685.393,E2 -11685.393} C_VEL
LIN {X 0,Y 390.148,Z 230.886,A -85,B 0,C 180,E1 -11688.571,E2 -11688.571} C_VEL
LIN {X 0,Y 390.307,Z 230.862,A -85,B 0,C 180,E1 -11692.032,E2 -11692.032} C_VEL
LIN {X 0,Y 390.224,Z 230.872,A -85,B 0,C 180,E1 -11694.834,E2 -11694.834} C_VEL
LIN {X 0,Y 390.42,Z 230.85,A -85,B 0,C 180,E1 -11697.937,E2 -11697.937} C_VEL
LIN {X 0,Y 390.547,Z 230.827,A -85,B 0,C 180,E1 -11700,E2 -11700} C_VEL
LIN {X 0,Y 390.312,Z 230.861,A -85,B 0,C 180,E1 -11703.097,E2 -11703.097} C_VEL
LIN {X 0,Y 390.308,Z 230.862,A -85,B 0,C 180,E1 -11706.594,E2 -11706.594} C_VEL
LIN {X 0,Y 390.314,Z 230.86,A -85,B 0,C 180,E1 -11708.282,E2 -11708.282} C_VEL
LIN {X 0,Y 390.17,Z 230.88,A -85,B 0,C 180,E1 -11712.483,E2 -11712.483} C_VEL
LIN {X 0,Y 390.139,Z 230.883,A -85,B 0,C 180,E1 -11715.677,E2 -11715.677} C_VEL
LIN {X 0,Y 390.105,Z 230.892,A -85,B 0,C 180,E1 -11718.922,E2 -11718.922} C_VEL
LIN {X 0,Y 390.037,Z 230.9,A -85,B 0,C 180,E1 -11722.234,E2 -11722.234} C_VEL
LIN {X 0,Y 390.084,Z 230.893,A -85,B 0,C 180,E1 -11725.733,E2 -11725.733} C_VEL
LIN {X 0,Y 390.043,Z 230.893,A -85,B 0,C 180,E1 -11729.111,E2 -11729.111} C_VEL
LIN {X 0,Y 390.043,Z 230.899,A -85,B 0,C 180,E1 -11732.722,E2 -11732.722} C_VEL
LIN {X 0,Y 390.054,Z 230.901,A -85,B 0,C 180,E1 -11735.825,E2 -11735.825} C_VEL
LIN {X 0,Y 390.036,Z 230.901,A -85,B 0,C 180,E1 -11739.212,E2 -11739.212} C_VEL
LIN {X 0,Y 390.059,Z 230.9,A -85,B 0,C 180,E1 -11740.664,E2 -11740.664} C_VEL
LIN {X 0,Y 392.213,Z 241.361,A -85,B 0,C 180,E1 -11743.267,E2 -11743.267} C_VEL
LIN {X 0,Y 392.688,Z 245.641,A -85,B 0,C 180,E1 -11744.284,E2 -11744.284} C_VEL
LIN {X 0,Y 392.676,Z 246.365,A -85,B 0,C 180,E1 -11744.429,E2 -11744.429} C_VEL
LIN {X 0,Y 397.518,Z 269.489,A -85,B 0,C 180,E1 -11745.165,E2 -11745.165} C_VEL
LIN {X 0,Y 396.132,Z 353.894,A -85,B 0,C 180,E1 -11746.757,E2 -11746.757} C_VEL
LIN {X 0,Y 395.647,Z 367.653,A -85,B 0,C 180,E1 -11747.232,E2 -11747.232} C_VEL
LIN {X 0,Y 394.99,Z 380.553,A -85,B 0,C 180,E1 -11747.897,E2 -11747.897} C_VEL
LIN {X 0,Y 394.198,Z 392.315,A -85,B 0,C 180,E1 -11748.726,E2 -11748.726} C_VEL
LIN {X 0,Y 393.313,Z 404.068,A -85,B 0,C 180,E1 -11749.796,E2 -11749.796} C_VEL
LIN {X 0,Y 392.336,Z 414.697,A -85,B 0,C 180,E1 -11751.019,E2 -11751.019} C_VEL
LIN {X 0,Y 391.425,Z 424.147,A -85,B 0,C 180,E1 -11752.377,E2 -11752.377} C_VEL
LIN {X 0,Y 390.642,Z 432.595,A -85,B 0,C 180,E1 -11753.878,E2 -11753.878} C_VEL
LIN {X 0,Y 389.961,Z 439.54,A -85,B 0,C 180,E1 -11755.41,E2 -11755.41} C_VEL
LIN {X 0,Y 389.431,Z 445.94,A -85,B 0,C 180,E1 -11757.221,E2 -11757.221} C_VEL
LIN {X 0,Y 389.068,Z 450.747,A -85,B 0,C 180,E1 -11759.015,E2 -11759.015} C_VEL
LIN {X 0,Y 388.772,Z 454.137,A -85,B 0,C 180,E1 -11760.785,E2 -11760.785} C_VEL
LIN {X 0,Y 388.571,Z 456.139,A -85,B 0,C 180,E1 -11762.407,E2 -11762.407} C_VEL
LIN {X 0,Y 388.454,Z 457.204,A -85,B 0,C 180,E1 -11764.265,E2 -11764.265} C_VEL
LIN {X 0,Y 388.443,Z 457.222,A -85,B 0,C 180,E1 -11765.409,E2 -11765.409} C_VEL
LIN {X 0,Y 388.516,Z 456.221,A -85,B 0,C 180,E1 -11767.303,E2 -11767.303} C_VEL
LIN {X 0,Y 388.681,Z 454.455,A -85,B 0,C 180,E1 -11768.799,E2 -11768.799} C_VEL
LIN {X 0,Y 388.936,Z 451.353,A -85,B 0,C 180,E1 -11770.522,E2 -11770.522} C_VEL
LIN {X 0,Y 389.193,Z 447.344,A -85,B 0,C 180,E1 -11772.122,E2 -11772.122} C_VEL
LIN {X 0,Y 389.584,Z 441.986,A -85,B 0,C 180,E1 -11773.763,E2 -11773.763} C_VEL
LIN {X 0,Y 390.168,Z 435.163,A -85,B 0,C 180,E1 -11775.393,E2 -11775.393} C_VEL
LIN {X 0,Y 390.904,Z 426.662,A -85,B 0,C 180,E1 -11777.013,E2 -11777.013} C_VEL
LIN {X 0,Y 391.678,Z 417.928,A -85,B 0,C 180,E1 -11778.354,E2 -11778.354} C_VEL
LIN {X 0,Y 392.584,Z 407.071,A -85,B 0,C 180,E1 -11779.687,E2 -11779.687} C_VEL
LIN {X 0,Y 393.409,Z 396.275,A -85,B 0,C 180,E1 -11780.748,E2 -11780.748} C_VEL
LIN {X 0,Y 394.11,Z 386.166,A -85,B 0,C 180,E1 -11781.54,E2 -11781.54} C_VEL
LIN {X 0,Y 394.739,Z 374.361,A -85,B 0,C 180,E1 -11782.262,E2 -11782.262} C_VEL
LIN {X 0,Y 395.281,Z 361.564,A -85,B 0,C 180,E1 -11782.818,E2 -11782.818} C_VEL
LIN {X 0,Y 395.663,Z 348.544,A -85,B 0,C 180,E1 -11783.176,E2 -11783.176} C_VEL
LIN {X 0,Y 396.685,Z 279.253,A -85,B 0,C 180,E1 -11784.456,E2 -11784.456} C_VEL
LIN {X 0,Y 396.334,Z 275.396,A -85,B 0,C 180,E1 -11784.547,E2 -11784.547} C_VEL
LIN {X 0,Y 395.337,Z 271.68,A -85,B 0,C 180,E1 -11784.668,E2 -11784.668} C_VEL
LIN {X 0,Y 392.204,Z 264.636,A -85,B 0,C 180,E1 -11784.961,E2 -11784.961} C_VEL
LIN {X 0,Y 388.657,Z 257.658,A -85,B 0,C 180,E1 -11785.279,E2 -11785.279} C_VEL
LIN {X 0,Y 386.59,Z 252.168,A -85,B 0,C 180,E1 -11785.495,E2 -11785.495} C_VEL
LIN {X 0,Y 386.136,Z 250.251,A -85,B 0,C 180,E1 -11785.557,E2 -11785.557} C_VEL
LIN {X 0,Y 385.411,Z 246.407,A -85,B 0,C 180,E1 -11785.686,E2 -11785.686} C_VEL
LIN {X 0,Y 384.865,Z 240.742,A -85,B 0,C 180,E1 -11787.121,E2 -11787.121} C_VEL
LIN {X 0,Y 383.306,Z 231.735,A -85,B 0,C 180,E1 -11789.54,E2 -11789.54} C_VEL
LIN {X 0,Y 383.377,Z 231.729,A -85,B 0,C 180,E1 -11792.101,E2 -11792.101} C_VEL
LIN {X 0,Y 383.242,Z 231.745,A -85,B 0,C 180,E1 -11796.317,E2 -11796.317} C_VEL
LIN {X 0,Y 383.145,Z 231.759,A -85,B 0,C 180,E1 -11799.502,E2 -11799.502} C_VEL
LIN {X 0,Y 383.128,Z 231.761,A -85,B 0,C 180,E1 -11803.536,E2 -11803.536} C_VEL
LIN {X 0,Y 383.097,Z 231.764,A -85,B 0,C 180,E1 -11807.454,E2 -11807.454} C_VEL
LIN {X 0,Y 383.031,Z 231.77,A -85,B 0,C 180,E1 -11810.647,E2 -11810.647} C_VEL
LIN {X 0,Y 383.023,Z 231.777,A -85,B 0,C 180,E1 -11813.808,E2 -11813.808} C_VEL
LIN {X 0,Y 382.995,Z 231.776,A -85,B 0,C 180,E1 -11817.306,E2 -11817.306} C_VEL
LIN {X 0,Y 382.983,Z 231.776,A -85,B 0,C 180,E1 -11820.918,E2 -11820.918} C_VEL
LIN {X 0,Y 383.018,Z 231.772,A -85,B 0,C 180,E1 -11824.667,E2 -11824.667} C_VEL
LIN {X 0,Y 382.997,Z 231.779,A -85,B 0,C 180,E1 -11827.903,E2 -11827.903} C_VEL
LIN {X 0,Y 382.972,Z 231.779,A -85,B 0,C 180,E1 -11831.348,E2 -11831.348} C_VEL
LIN {X 0,Y 382.995,Z 231.778,A -85,B 0,C 180,E1 -11834.303,E2 -11834.303} C_VEL
LIN {X 0,Y 383.009,Z 231.774,A -85,B 0,C 180,E1 -11837.24,E2 -11837.24} C_VEL
LIN {X 0,Y 383.013,Z 231.775,A -85,B 0,C 180,E1 -11840.413,E2 -11840.413} C_VEL
LIN {X 0,Y 383.024,Z 231.775,A -85,B 0,C 180,E1 -11844.044,E2 -11844.044} C_VEL
LIN {X 0,Y 382.985,Z 231.778,A -85,B 0,C 180,E1 -11847.578,E2 -11847.578} C_VEL
LIN {X 0,Y 382.99,Z 231.779,A -85,B 0,C 180,E1 -11850.3,E2 -11850.3} C_VEL
LIN {X 0,Y 383.078,Z 231.769,A -85,B 0,C 180,E1 -11854.02,E2 -11854.02} C_VEL
LIN {X 0,Y 383.006,Z 231.774,A -85,B 0,C 180,E1 -11857.335,E2 -11857.335} C_VEL
LIN {X 0,Y 383.058,Z 231.768,A -85,B 0,C 180,E1 -11860.716,E2 -11860.716} C_VEL
LIN {X 0,Y 383.078,Z 231.769,A -85,B 0,C 180,E1 -11864.026,E2 -11864.026} C_VEL
LIN {X 0,Y 383.134,Z 231.758,A -85,B 0,C 180,E1 -11867.284,E2 -11867.284} C_VEL
LIN {X 0,Y 383.149,Z 231.759,A -85,B 0,C 180,E1 -11870.498,E2 -11870.498} C_VEL
LIN {X 0,Y 383.271,Z 231.743,A -85,B 0,C 180,E1 -11872.625,E2 -11872.625} C_VEL
LIN {X 0,Y 383.197,Z 231.751,A -85,B 0,C 180,E1 -11874.738,E2 -11874.738} C_VEL
LIN {X 0,Y 383.385,Z 231.73,A -85,B 0,C 180,E1 -11877.899,E2 -11877.899} C_VEL
LIN {X 0,Y 383.515,Z 231.714,A -85,B 0,C 180,E1 -11880,E2 -11880} C_VEL
LIN {X 0,Y 383.249,Z 231.743,A -85,B 0,C 180,E1 -11883.154,E2 -11883.154} C_VEL
LIN {X 0,Y 383.285,Z 231.743,A -85,B 0,C 180,E1 -11886.316,E2 -11886.316} C_VEL
LIN {X 0,Y 383.257,Z 231.747,A -85,B 0,C 180,E1 -11888.436,E2 -11888.436} C_VEL
LIN {X 0,Y 383.095,Z 231.764,A -85,B 0,C 180,E1 -11891.642,E2 -11891.642} C_VEL
LIN {X 0,Y 383.107,Z 231.762,A -85,B 0,C 180,E1 -11894.882,E2 -11894.882} C_VEL
LIN {X 0,Y 383.087,Z 231.767,A -85,B 0,C 180,E1 -11898.172,E2 -11898.172} C_VEL
LIN {X 0,Y 382.991,Z 231.776,A -85,B 0,C 180,E1 -11901.531,E2 -11901.531} C_VEL
LIN {X 0,Y 383.05,Z 231.769,A -85,B 0,C 180,E1 -11904.96,E2 -11904.96} C_VEL
LIN {X 0,Y 383.038,Z 231.774,A -85,B 0,C 180,E1 -11908.493,E2 -11908.493} C_VEL
LIN {X 0,Y 383.007,Z 231.777,A -85,B 0,C 180,E1 -11912.15,E2 -11912.15} C_VEL
LIN {X 0,Y 383.016,Z 231.775,A -85,B 0,C 180,E1 -11914.668,E2 -11914.668} C_VEL
LIN {X 0,Y 382.997,Z 231.776,A -85,B 0,C 180,E1 -11917.904,E2 -11917.904} C_VEL
LIN {X 0,Y 382.982,Z 231.776,A -85,B 0,C 180,E1 -11921.348,E2 -11921.348} C_VEL
LIN {X 0,Y 382.994,Z 231.779,A -85,B 0,C 180,E1 -11924.304,E2 -11924.304} C_VEL
LIN {X 0,Y 383.009,Z 231.773,A -85,B 0,C 180,E1 -11927.241,E2 -11927.241} C_VEL
LIN {X 0,Y 383.014,Z 231.777,A -85,B 0,C 180,E1 -11930.414,E2 -11930.414} C_VEL
LIN {X 0,Y 383.024,Z 231.773,A -85,B 0,C 180,E1 -11934.045,E2 -11934.045} C_VEL
LIN {X 0,Y 382.987,Z 231.778,A -85,B 0,C 180,E1 -11937.578,E2 -11937.578} C_VEL
LIN {X 0,Y 383.082,Z 231.824,A -85,B 0,C 180,E1 -11941.399,E2 -11941.399} C_VEL
LIN {X 0,Y 385.262,Z 242.594,A -85,B 0,C 180,E1 -11944.036,E2 -11944.036} C_VEL
LIN {X 0,Y 386.347,Z 248.508,A -85,B 0,C 180,E1 -11945.443,E2 -11945.443} C_VEL
LIN {X 0,Y 386.091,Z 254.07,A -85,B 0,C 180,E1 -11946.677,E2 -11946.677} C_VEL
LIN {X 0,Y 385.084,Z 266.419,A -85,B 0,C 180,E1 -11949.345,E2 -11949.345} C_VEL
LIN {X 0,Y 389.796,Z 296.406,A -85,B 0,C 180,E1 -11950.176,E2 -11950.176} C_VEL
LIN {X 0,Y 388.589,Z 375.158,A -85,B 0,C 180,E1 -11951.685,E2 -11951.685} C_VEL
LIN {X 0,Y 388.006,Z 388.886,A -85,B 0,C 180,E1 -11952.168,E2 -11952.168} C_VEL
LIN {X 0,Y 387.285,Z 400.716,A -85,B 0,C 180,E1 -11952.782,E2 -11952.782} C_VEL
LIN {X 0,Y 386.412,Z 412.726,A -85,B 0,C 180,E1 -11953.626,E2 -11953.626} C_VEL
LIN {X 0,Y 385.493,Z 424.225,A -85,B 0,C 180,E1 -11954.672,E2 -11954.672} C_VEL
LIN {X 0,Y 384.669,Z 434.781,A -85,B 0,C 180,E1 -11955.879,E2 -11955.879} C_VEL
LIN {X 0,Y 383.937,Z 443.073,A -85,B 0,C 180,E1 -11957.042,E2 -11957.042} C_VEL
LIN {X 0,Y 382.981,Z 452.246,A -85,B 0,C 180,E1 -11958.623,E2 -11958.623} C_VEL
LIN {X 0,Y 382.421,Z 459.64,A -85,B 0,C 180,E1 -11960.213,E2 -11960.213} C_VEL
LIN {X 0,Y 382.061,Z 464.652,A -85,B 0,C 180,E1 -11961.538,E2 -11961.538} C_VEL
LIN {X 0,Y 381.784,Z 469.512,A -85,B 0,C 180,E1 -11963.128,E2 -11963.128} C_VEL
LIN {X 0,Y 381.64,Z 473.24,A -85,B 0,C 180,E1 -11964.717,E2 -11964.717} C_VEL
LIN {X 0,Y 381.624,Z 475.163,A -85,B 0,C 180,E1 -11965.776,E2 -11965.776} C_VEL
LIN {X 0,Y 381.547,Z 476.643,A -85,B 0,C 180,E1 -11966.832,E2 -11966.832} C_VEL
LIN {X 0,Y 381.617,Z 478.328,A -85,B 0,C 180,E1 -11968.945,E2 -11968.945} C_VEL
LIN {X 0,Y 381.639,Z 478.584,A -85,B 0,C 180,E1 -11970,E2 -11970} C_VEL
LIN {X 0,Y 381.602,Z 478.429,A -85,B 0,C 180,E1 -11971.055,E2 -11971.055} C_VEL
LIN {X 0,Y 381.546,Z 476.874,A -85,B 0,C 180,E1 -11973.168,E2 -11973.168} C_VEL
LIN {X 0,Y 381.624,Z 475.506,A -85,B 0,C 180,E1 -11974.225,E2 -11974.225} C_VEL
LIN {X 0,Y 381.67,Z 472.01,A -85,B 0,C 180,E1 -11976.094,E2 -11976.094} C_VEL
LIN {X 0,Y 381.952,Z 467.133,A -85,B 0,C 180,E1 -11977.932,E2 -11977.932} C_VEL
LIN {X 0,Y 382.466,Z 460.646,A -85,B 0,C 180,E1 -11979.786,E2 -11979.786} C_VEL
LIN {X 0,Y 383.051,Z 453.555,A -85,B 0,C 180,E1 -11981.375,E2 -11981.375} C_VEL
LIN {X 0,Y 384.009,Z 444.705,A -85,B 0,C 180,E1 -11982.956,E2 -11982.956} C_VEL
LIN {X 0,Y 384.873,Z 435.358,A -85,B 0,C 180,E1 -11984.311,E2 -11984.311} C_VEL
LIN {X 0,Y 385.713,Z 425.694,A -85,B 0,C 180,E1 -11985.455,E2 -11985.455} C_VEL
LIN {X 0,Y 386.732,Z 414.661,A -85,B 0,C 180,E1 -11986.496,E2 -11986.496} C_VEL
LIN {X 0,Y 387.717,Z 402.321,A -85,B 0,C 180,E1 -11987.403,E2 -11987.403} C_VEL
LIN {X 0,Y 388.563,Z 390.647,A -85,B 0,C 180,E1 -11988.044,E2 -11988.044} C_VEL
LIN {X 0,Y 389.171,Z 378.188,A -85,B 0,C 180,E1 -11988.525,E2 -11988.525} C_VEL
LIN {X 0,Y 389.641,Z 360.837,A -85,B 0,C 180,E1 -11988.911,E2 -11988.911} C_VEL
LIN {X 0,Y 390.48,Z 295.819,A -85,B 0,C 180,E1 -11990.152,E2 -11990.152} C_VEL
LIN {X 0,Y 386.259,Z 270.227,A -85,B 0,C 180,E1 -11990.913,E2 -11990.913} C_VEL
LIN {X 0,Y 385.344,Z 265.511,A -85,B 0,C 180,E1 -11991.085,E2 -11991.085} C_VEL
LIN {X 0,Y 386.512,Z 251.429,A -85,B 0,C 180,E1 -11994.121,E2 -11994.121} C_VEL
LIN {X 0,Y 386.275,Z 247.452,A -85,B 0,C 180,E1 -11995.025,E2 -11995.025} C_VEL
LIN {X 0,Y 384.019,Z 235.883,A -85,B 0,C 180,E1 -11997.819,E2 -11997.819} C_VEL
LIN {X 0,Y 383.064,Z 231.767,A -85,B 0,C 180,E1 -11998.865,E2 -11998.865} C_VEL
LIN {X 0,Y 382.988,Z 231.782,A -85,B 0,C 180,E1 -12002.422,E2 -12002.422} C_VEL
LIN {X 0,Y 383.025,Z 231.773,A -85,B 0,C 180,E1 -12005.955,E2 -12005.955} C_VEL
LIN {X 0,Y 383.015,Z 231.774,A -85,B 0,C 180,E1 -12009.586,E2 -12009.586} C_VEL
LIN {X 0,Y 383.005,Z 231.774,A -85,B 0,C 180,E1 -12012.778,E2 -12012.778} C_VEL
LIN {X 0,Y 382.998,Z 231.778,A -85,B 0,C 180,E1 -12015.789,E2 -12015.789} C_VEL
LIN {X 0,Y 382.988,Z 231.775,A -85,B 0,C 180,E1 -12018.796,E2 -12018.796} C_VEL
LIN {X 0,Y 382.999,Z 231.773,A -85,B 0,C 180,E1 -12022.096,E2 -12022.096} C_VEL
LIN {X 0,Y 383.018,Z 231.772,A -85,B 0,C 180,E1 -12025.332,E2 -12025.332} C_VEL
LIN {X 0,Y 382.982,Z 231.774,A -85,B 0,C 180,E1 -12029.081,E2 -12029.081} C_VEL
LIN {X 0,Y 383.056,Z 231.764,A -85,B 0,C 180,E1 -12032.698,E2 -12032.698} C_VEL
LIN {X 0,Y 383.052,Z 231.773,A -85,B 0,C 180,E1 -12035.04,E2 -12035.04} C_VEL
LIN {X 0,Y 382.992,Z 231.775,A -85,B 0,C 180,E1 -12038.469,E2 -12038.469} C_VEL
LIN {X 0,Y 383.089,Z 231.759,A -85,B 0,C 180,E1 -12041.828,E2 -12041.828} C_VEL
LIN {X 0,Y 383.11,Z 231.757,A -85,B 0,C 180,E1 -12045.118,E2 -12045.118} C_VEL
LIN {X 0,Y 383.097,Z 231.763,A -85,B 0,C 180,E1 -12048.358,E2 -12048.358} C_VEL
LIN {X 0,Y 383.263,Z 231.74,A -85,B 0,C 180,E1 -12051.976,E2 -12051.976} C_VEL
LIN {X 0,Y 383.196,Z 231.748,A -85,B 0,C 180,E1 -12054.739,E2 -12054.739} C_VEL
LIN {X 0,Y 383.387,Z 231.726,A -85,B 0,C 180,E1 -12057.899,E2 -12057.899} C_VEL
LIN {X 0,Y 383.517,Z 231.703,A -85,B 0,C 180,E1 -12060,E2 -12060} C_VEL
LIN {X 0,Y 383.248,Z 231.741,A -85,B 0,C 180,E1 -12063.154,E2 -12063.154} C_VEL
LIN {X 0,Y 383.269,Z 231.74,A -85,B 0,C 180,E1 -12066.587,E2 -12066.587} C_VEL
LIN {X 0,Y 383.26,Z 231.739,A -85,B 0,C 180,E1 -12068.436,E2 -12068.436} C_VEL
LIN {X 0,Y 383.097,Z 231.757,A -85,B 0,C 180,E1 -12071.642,E2 -12071.642} C_VEL
LIN {X 0,Y 383.11,Z 231.76,A -85,B 0,C 180,E1 -12074.882,E2 -12074.882} C_VEL
LIN {X 0,Y 383.089,Z 231.764,A -85,B 0,C 180,E1 -12078.172,E2 -12078.172} C_VEL
LIN {X 0,Y 382.992,Z 231.775,A -85,B 0,C 180,E1 -12081.531,E2 -12081.531} C_VEL
LIN {X 0,Y 383.028,Z 231.775,A -85,B 0,C 180,E1 -12084.962,E2 -12084.962} C_VEL
LIN {X 0,Y 383.002,Z 231.772,A -85,B 0,C 180,E1 -12088.496,E2 -12088.496} C_VEL
LIN {X 0,Y 383.009,Z 231.773,A -85,B 0,C 180,E1 -12092.15,E2 -12092.15} C_VEL
LIN {X 0,Y 383.017,Z 231.776,A -85,B 0,C 180,E1 -12094.668,E2 -12094.668} C_VEL
LIN {X 0,Y 382.992,Z 231.78,A -85,B 0,C 180,E1 -12097.902,E2 -12097.902} C_VEL
LIN {X 0,Y 383.032,Z 231.868,A -85,B 0,C 180,E1 -12100.343,E2 -12100.343} C_VEL
LIN {X 0,Y 385.52,Z 243.886,A -85,B 0,C 180,E1 -12103.385,E2 -12103.385} C_VEL
LIN {X 0,Y 385.819,Z 246.573,A -85,B 0,C 180,E1 -12104.017,E2 -12104.017} C_VEL
LIN {X 0,Y 390.786,Z 269.9,A -85,B 0,C 180,E1 -12104.787,E2 -12104.787} C_VEL
LIN {X 0,Y 390.849,Z 276.75,A -85,B 0,C 180,E1 -12104.927,E2 -12104.927} C_VEL
LIN {X 0,Y 389.443,Z 354.26,A -85,B 0,C 180,E1 -12106.414,E2 -12106.414} C_VEL
LIN {X 0,Y 388.933,Z 368.052,A -85,B 0,C 180,E1 -12106.9,E2 -12106.9} C_VEL
LIN {X 0,Y 388.316,Z 379.963,A -85,B 0,C 180,E1 -12107.522,E2 -12107.522} C_VEL
LIN {X 0,Y 387.485,Z 392.024,A -85,B 0,C 180,E1 -12108.373,E2 -12108.373} C_VEL
LIN {X 0,Y 386.615,Z 402.771,A -85,B 0,C 180,E1 -12109.348,E2 -12109.348} C_VEL
LIN {X 0,Y 385.654,Z 413.285,A -85,B 0,C 180,E1 -12110.539,E2 -12110.539} C_VEL
LIN {X 0,Y 384.722,Z 422.114,A -85,B 0,C 180,E1 -12111.769,E2 -12111.769} C_VEL
LIN {X 0,Y 383.841,Z 431.128,A -85,B 0,C 180,E1 -12113.329,E2 -12113.329} C_VEL
LIN {X 0,Y 383.053,Z 438.917,A -85,B 0,C 180,E1 -12115.016,E2 -12115.016} C_VEL
LIN {X 0,Y 382.491,Z 444.553,A -85,B 0,C 180,E1 -12116.549,E2 -12116.549} C_VEL
LIN {X 0,Y 382.099,Z 449.782,A -85,B 0,C 180,E1 -12118.385,E2 -12118.385} C_VEL
LIN {X 0,Y 381.789,Z 453.518,A -85,B 0,C 180,E1 -12120.197,E2 -12120.197} C_VEL
LIN {X 0,Y 381.494,Z 456.154,A -85,B 0,C 180,E1 -12122.162,E2 -12122.162} C_VEL
LIN {X 0,Y 381.386,Z 457.239,A -85,B 0,C 180,E1 -12123.752,E2 -12123.752} C_VEL
LIN {X 0,Y 381.366,Z 457.49,A -85,B 0,C 180,E1 -12124.922,E2 -12124.922} C_VEL
LIN {X 0,Y 381.336,Z 457.214,A -85,B 0,C 180,E1 -12126.08,E2 -12126.08} C_VEL
LIN {X 0,Y 381.419,Z 456.487,A -85,B 0,C 180,E1 -12127.236,E2 -12127.236} C_VEL
LIN {X 0,Y 381.519,Z 455.298,A -85,B 0,C 180,E1 -12128.382,E2 -12128.382} C_VEL
LIN {X 0,Y 381.74,Z 452.998,A -85,B 0,C 180,E1 -12129.874,E2 -12129.874} C_VEL
LIN {X 0,Y 382.072,Z 448.767,A -85,B 0,C 180,E1 -12131.778,E2 -12131.778} C_VEL
LIN {X 0,Y 382.413,Z 443.669,A -85,B 0,C 180,E1 -12133.473,E2 -12133.473} C_VEL
LIN {X 0,Y 382.963,Z 437.366,A -85,B 0,C 180,E1 -12135.112,E2 -12135.112} C_VEL
LIN {X 0,Y 383.672,Z 429.356,A -85,B 0,C 180,E1 -12136.77,E2 -12136.77} C_VEL
LIN {X 0,Y 384.455,Z 421.149,A -85,B 0,C 180,E1 -12138.132,E2 -12138.132} C_VEL
LIN {X 0,Y 385.326,Z 411.09,A -85,B 0,C 180,E1 -12139.491,E2 -12139.491} C_VEL
LIN {X 0,Y 386.169,Z 401.178,A -85,B 0,C 180,E1 -12140.573,E2 -12140.573} C_VEL
LIN {X 0,Y 387.081,Z 390.381,A -85,B 0,C 180,E1 -12141.517,E2 -12141.517} C_VEL
LIN {X 0,Y 387.748,Z 378.631,A -85,B 0,C 180,E1 -12142.318,E2 -12142.318} C_VEL
LIN {X 0,Y 388.329,Z 365.554,A -85,B 0,C 180,E1 -12142.973,E2 -12142.973} C_VEL
LIN {X 0,Y 388.756,Z 352.906,A -85,B 0,C 180,E1 -12143.392,E2 -12143.392} C_VEL
LIN {X 0,Y 390.013,Z 269.666,A -85,B 0,C 180,E1 -12144.973,E2 -12144.973} C_VEL
LIN {X 0,Y 386.136,Z 250.251,A -85,B 0,C 180,E1 -12145.557,E2 -12145.557} C_VEL
LIN {X 0,Y 385.3,Z 247.628,A -85,B 0,C 180,E1 -12145.734,E2 -12145.734} C_VEL
LIN {X 0,Y 383.796,Z 245.122,A -85,B 0,C 180,E1 -12146.126,E2 -12146.126} C_VEL
LIN {X 0,Y 379.384,Z 240.27,A -85,B 0,C 180,E1 -12147.624,E2 -12147.624} C_VEL
LIN {X 0,Y 377.14,Z 236.213,A -85,B 0,C 180,E1 -12148.784,E2 -12148.784} C_VEL
LIN {X 0,Y 376.535,Z 234.046,A -85,B 0,C 180,E1 -12149.373,E2 -12149.373} C_VEL
LIN {X 0,Y 376.28,Z 232.61,A -85,B 0,C 180,E1 -12149.799,E2 -12149.799} C_VEL
LIN {X 0,Y 376.342,Z 232.606,A -85,B 0,C 180,E1 -12152.14,E2 -12152.14} C_VEL
LIN {X 0,Y 376.201,Z 232.621,A -85,B 0,C 180,E1 -12156.436,E2 -12156.436} C_VEL
LIN {X 0,Y 376.116,Z 232.637,A -85,B 0,C 180,E1 -12159.681,E2 -12159.681} C_VEL
LIN {X 0,Y 376.092,Z 232.639,A -85,B 0,C 180,E1 -12163.657,E2 -12163.657} C_VEL
LIN {X 0,Y 376.045,Z 232.644,A -85,B 0,C 180,E1 -12167.606,E2 -12167.606} C_VEL
LIN {X 0,Y 375.98,Z 232.648,A -85,B 0,C 180,E1 -12170.832,E2 -12170.832} C_VEL
LIN {X 0,Y 375.981,Z 232.65,A -85,B 0,C 180,E1 -12174.282,E2 -12174.282} C_VEL
LIN {X 0,Y 375.937,Z 232.659,A -85,B 0,C 180,E1 -12177.863,E2 -12177.863} C_VEL
LIN {X 0,Y 375.958,Z 232.654,A -85,B 0,C 180,E1 -12181.561,E2 -12181.561} C_VEL
LIN {X 0,Y 375.957,Z 232.653,A -85,B 0,C 180,E1 -12185.415,E2 -12185.415} C_VEL
LIN {X 0,Y 375.97,Z 232.653,A -85,B 0,C 180,E1 -12188.269,E2 -12188.269} C_VEL
LIN {X 0,Y 375.925,Z 232.658,A -85,B 0,C 180,E1 -12191.599,E2 -12191.599} C_VEL
LIN {X 0,Y 375.926,Z 232.656,A -85,B 0,C 180,E1 -12195.268,E2 -12195.268} C_VEL
LIN {X 0,Y 375.933,Z 232.657,A -85,B 0,C 180,E1 -12198.399,E2 -12198.399} C_VEL
LIN {X 0,Y 375.972,Z 232.653,A -85,B 0,C 180,E1 -12201.729,E2 -12201.729} C_VEL
LIN {X 0,Y 375.979,Z 232.649,A -85,B 0,C 180,E1 -12205.332,E2 -12205.332} C_VEL
LIN {X 0,Y 375.956,Z 232.654,A -85,B 0,C 180,E1 -12208.438,E2 -12208.438} C_VEL
LIN {X 0,Y 375.982,Z 232.653,A -85,B 0,C 180,E1 -12212.14,E2 -12212.14} C_VEL
LIN {X 0,Y 376.004,Z 232.647,A -85,B 0,C 180,E1 -12214.539,E2 -12214.539} C_VEL
LIN {X 0,Y 375.961,Z 232.656,A -85,B 0,C 180,E1 -12218.045,E2 -12218.045} C_VEL
LIN {X 0,Y 376.021,Z 232.644,A -85,B 0,C 180,E1 -12221.474,E2 -12221.474} C_VEL
LIN {X 0,Y 376.056,Z 232.64,A -85,B 0,C 180,E1 -12224.832,E2 -12224.832} C_VEL
LIN {X 0,Y 376.048,Z 232.645,A -85,B 0,C 180,E1 -12228.136,E2 -12228.136} C_VEL
LIN {X 0,Y 376.255,Z 232.618,A -85,B 0,C 180,E1 -12231.877,E2 -12231.877} C_VEL
LIN {X 0,Y 376.169,Z 232.627,A -85,B 0,C 180,E1 -12234.64,E2 -12234.64} C_VEL
LIN {X 0,Y 376.351,Z 232.606,A -85,B 0,C 180,E1 -12237.86,E2 -12237.86} C_VEL
LIN {X 0,Y 376.484,Z 232.59,A -85,B 0,C 180,E1 -12240,E2 -12240} C_VEL
LIN {X 0,Y 376.187,Z 232.623,A -85,B 0,C 180,E1 -12243.213,E2 -12243.213} C_VEL
LIN {X 0,Y 376.244,Z 232.62,A -85,B 0,C 180,E1 -12246.435,E2 -12246.435} C_VEL
LIN {X 0,Y 376.203,Z 232.624,A -85,B 0,C 180,E1 -12248.595,E2 -12248.595} C_VEL
LIN {X 0,Y 376.047,Z 232.643,A -85,B 0,C 180,E1 -12251.863,E2 -12251.863} C_VEL
LIN {X 0,Y 376.056,Z 232.639,A -85,B 0,C 180,E1 -12255.168,E2 -12255.168} C_VEL
LIN {X 0,Y 376.021,Z 232.647,A -85,B 0,C 180,E1 -12258.526,E2 -12258.526} C_VEL
LIN {X 0,Y 375.961,Z 232.654,A -85,B 0,C 180,E1 -12261.954,E2 -12261.954} C_VEL
LIN {X 0,Y 376.004,Z 232.645,A -85,B 0,C 180,E1 -12265.461,E2 -12265.461} C_VEL
LIN {X 0,Y 375.968,Z 232.65,A -85,B 0,C 180,E1 -12269.079,E2 -12269.079} C_VEL
LIN {X 0,Y 375.947,Z 232.654,A -85,B 0,C 180,E1 -12272.829,E2 -12272.829} C_VEL
LIN {X 0,Y 375.956,Z 232.651,A -85,B 0,C 180,E1 -12275.416,E2 -12275.416} C_VEL
LIN {X 0,Y 375.972,Z 232.654,A -85,B 0,C 180,E1 -12278.271,E2 -12278.271} C_VEL
LIN {X 0,Y 375.932,Z 232.654,A -85,B 0,C 180,E1 -12281.601,E2 -12281.601} C_VEL
LIN {X 0,Y 375.925,Z 232.655,A -85,B 0,C 180,E1 -12285.269,E2 -12285.269} C_VEL
LIN {X 0,Y 375.934,Z 232.659,A -85,B 0,C 180,E1 -12288.4,E2 -12288.4} C_VEL
LIN {X 0,Y 375.973,Z 232.649,A -85,B 0,C 180,E1 -12291.73,E2 -12291.73} C_VEL
LIN {X 0,Y 375.979,Z 232.648,A -85,B 0,C 180,E1 -12295.333,E2 -12295.333} C_VEL
LIN {X 0,Y 375.958,Z 232.657,A -85,B 0,C 180,E1 -12298.438,E2 -12298.438} C_VEL
LIN {X 0,Y 376.035,Z 232.77,A -85,B 0,C 180,E1 -12301.118,E2 -12301.118} C_VEL
LIN {X 0,Y 378.244,Z 243.55,A -85,B 0,C 180,E1 -12303.814,E2 -12303.814} C_VEL
LIN {X 0,Y 379.437,Z 250.936,A -85,B 0,C 180,E1 -12305.594,E2 -12305.594} C_VEL
LIN {X 0,Y 378.372,Z 263.42,A -85,B 0,C 180,E1 -12308.375,E2 -12308.375} C_VEL
LIN {X 0,Y 378.169,Z 266.108,A -85,B 0,C 180,E1 -12308.971,E2 -12308.971} C_VEL
LIN {X 0,Y 383.012,Z 296.614,A -85,B 0,C 180,E1 -12309.84,E2 -12309.84} C_VEL
LIN {X 0,Y 381.842,Z 374.224,A -85,B 0,C 180,E1 -12311.35,E2 -12311.35} C_VEL
LIN {X 0,Y 381.272,Z 387.431,A -85,B 0,C 180,E1 -12311.808,E2 -12311.808} C_VEL
LIN {X 0,Y 380.489,Z 400.151,A -85,B 0,C 180,E1 -12312.464,E2 -12312.464} C_VEL
LIN {X 0,Y 379.588,Z 412.271,A -85,B 0,C 180,E1 -12313.323,E2 -12313.323} C_VEL
LIN {X 0,Y 378.609,Z 423.817,A -85,B 0,C 180,E1 -12314.386,E2 -12314.386} C_VEL
LIN {X 0,Y 377.838,Z 433.199,A -85,B 0,C 180,E1 -12315.463,E2 -12315.463} C_VEL
LIN {X 0,Y 376.987,Z 442.737,A -85,B 0,C 180,E1 -12316.799,E2 -12316.799} C_VEL
LIN {X 0,Y 375.99,Z 451.942,A -85,B 0,C 180,E1 -12318.408,E2 -12318.408} C_VEL
LIN {X 0,Y 375.393,Z 459.355,A -85,B 0,C 180,E1 -12320.028,E2 -12320.028} C_VEL
LIN {X 0,Y 374.885,Z 466.158,A -85,B 0,C 180,E1 -12321.917,E2 -12321.917} C_VEL
LIN {X 0,Y 374.631,Z 470.64,A -85,B 0,C 180,E1 -12323.537,E2 -12323.537} C_VEL
LIN {X 0,Y 374.551,Z 473.003,A -85,B 0,C 180,E1 -12324.617,E2 -12324.617} C_VEL
LIN {X 0,Y 374.55,Z 474.933,A -85,B 0,C 180,E1 -12325.696,E2 -12325.696} C_VEL
LIN {X 0,Y 374.461,Z 476.425,A -85,B 0,C 180,E1 -12326.772,E2 -12326.772} C_VEL
LIN {X 0,Y 374.517,Z 478.122,A -85,B 0,C 180,E1 -12328.925,E2 -12328.925} C_VEL
LIN {X 0,Y 374.554,Z 478.384,A -85,B 0,C 180,E1 -12330,E2 -12330} C_VEL
LIN {X 0,Y 374.502,Z 478.24,A -85,B 0,C 180,E1 -12331.075,E2 -12331.075} C_VEL
LIN {X 0,Y 374.46,Z 476.695,A -85,B 0,C 180,E1 -12333.228,E2 -12333.228} C_VEL
LIN {X 0,Y 374.528,Z 475.332,A -85,B 0,C 180,E1 -12334.305,E2 -12334.305} C_VEL
LIN {X 0,Y 374.566,Z 472.212,A -85,B 0,C 180,E1 -12336.042,E2 -12336.042} C_VEL
LIN {X 0,Y 374.797,Z 468.541,A -85,B 0,C 180,E1 -12337.543,E2 -12337.543} C_VEL
LIN {X 0,Y 375.19,Z 463.499,A -85,B 0,C 180,E1 -12339.162,E2 -12339.162} C_VEL
LIN {X 0,Y 375.739,Z 457.18,A -85,B 0,C 180,E1 -12340.78,E2 -12340.78} C_VEL
LIN {X 0,Y 376.579,Z 449.278,A -85,B 0,C 180,E1 -12342.393,E2 -12342.393} C_VEL
LIN {X 0,Y 377.416,Z 441.234,A -85,B 0,C 180,E1 -12343.735,E2 -12343.735} C_VEL
LIN {X 0,Y 378.307,Z 431.432,A -85,B 0,C 180,E1 -12345.075,E2 -12345.075} C_VEL
LIN {X 0,Y 379.392,Z 420.531,A -85,B 0,C 180,E1 -12346.271,E2 -12346.271} C_VEL
LIN {X 0,Y 380.359,Z 409.873,A -85,B 0,C 180,E1 -12347.196,E2 -12347.196} C_VEL
LIN {X 0,Y 381.377,Z 397.073,A -85,B 0,C 180,E1 -12348.048,E2 -12348.048} C_VEL
LIN {X 0,Y 382.158,Z 384.196,A -85,B 0,C 180,E1 -12348.669,E2 -12348.669} C_VEL
LIN {X 0,Y 382.734,Z 371.584,A -85,B 0,C 180,E1 -12349.057,E2 -12349.057} C_VEL
LIN {X 0,Y 383.894,Z 296.789,A -85,B 0,C 180,E1 -12350.515,E2 -12350.515} C_VEL
LIN {X 0,Y 379.739,Z 271.53,A -85,B 0,C 180,E1 -12351.286,E2 -12351.286} C_VEL
LIN {X 0,Y 378.512,Z 265.308,A -85,B 0,C 180,E1 -12351.511,E2 -12351.511} C_VEL
LIN {X 0,Y 379.669,Z 251.957,A -85,B 0,C 180,E1 -12354.446,E2 -12354.446} C_VEL
LIN {X 0,Y 378.829,Z 246.084,A -85,B 0,C 180,E1 -12355.847,E2 -12355.847} C_VEL
LIN {X 0,Y 376.915,Z 236.563,A -85,B 0,C 180,E1 -12358.21,E2 -12358.21} C_VEL
LIN {X 0,Y 376.005,Z 232.647,A -85,B 0,C 180,E1 -12359.229,E2 -12359.229} C_VEL
LIN {X 0,Y 375.95,Z 232.658,A -85,B 0,C 180,E1 -12362.828,E2 -12362.828} C_VEL
LIN {X 0,Y 375.958,Z 232.657,A -85,B 0,C 180,E1 -12365.415,E2 -12365.415} C_VEL
LIN {X 0,Y 375.973,Z 232.65,A -85,B 0,C 180,E1 -12368.27,E2 -12368.27} C_VEL
LIN {X 0,Y 375.936,Z 232.657,A -85,B 0,C 180,E1 -12371.601,E2 -12371.601} C_VEL
LIN {X 0,Y 375.928,Z 232.657,A -85,B 0,C 180,E1 -12375.268,E2 -12375.268} C_VEL
LIN {X 0,Y 375.934,Z 232.652,A -85,B 0,C 180,E1 -12378.399,E2 -12378.399} C_VEL
LIN {X 0,Y 375.973,Z 232.65,A -85,B 0,C 180,E1 -12381.73,E2 -12381.73} C_VEL
LIN {X 0,Y 375.98,Z 232.648,A -85,B 0,C 180,E1 -12385.333,E2 -12385.333} C_VEL
LIN {X 0,Y 375.957,Z 232.648,A -85,B 0,C 180,E1 -12388.438,E2 -12388.438} C_VEL
LIN {X 0,Y 375.983,Z 232.644,A -85,B 0,C 180,E1 -12392.14,E2 -12392.14} C_VEL
LIN {X 0,Y 376.006,Z 232.646,A -85,B 0,C 180,E1 -12394.539,E2 -12394.539} C_VEL
LIN {X 0,Y 375.963,Z 232.649,A -85,B 0,C 180,E1 -12398.046,E2 -12398.046} C_VEL
LIN {X 0,Y 376.023,Z 232.639,A -85,B 0,C 180,E1 -12401.474,E2 -12401.474} C_VEL
LIN {X 0,Y 376.058,Z 232.639,A -85,B 0,C 180,E1 -12404.833,E2 -12404.833} C_VEL
LIN {X 0,Y 376.049,Z 232.64,A -85,B 0,C 180,E1 -12408.137,E2 -12408.137} C_VEL
LIN {X 0,Y 376.218,Z 232.617,A -85,B 0,C 180,E1 -12411.919,E2 -12411.919} C_VEL
LIN {X 0,Y 376.169,Z 232.623,A -85,B 0,C 180,E1 -12414.64,E2 -12414.64} C_VEL
LIN {X 0,Y 376.353,Z 232.602,A -85,B 0,C 180,E1 -12417.86,E2 -12417.86} C_VEL
LIN {X 0,Y 376.486,Z 232.579,A -85,B 0,C 180,E1 -12420,E2 -12420} C_VEL
LIN {X 0,Y 376.186,Z 232.62,A -85,B 0,C 180,E1 -12423.213,E2 -12423.213} C_VEL
LIN {X 0,Y 376.234,Z 232.618,A -85,B 0,C 180,E1 -12426.578,E2 -12426.578} C_VEL
LIN {X 0,Y 376.205,Z 232.619,A -85,B 0,C 180,E1 -12428.595,E2 -12428.595} C_VEL
LIN {X 0,Y 376.049,Z 232.635,A -85,B 0,C 180,E1 -12431.864,E2 -12431.864} C_VEL
LIN {X 0,Y 376.058,Z 232.638,A -85,B 0,C 180,E1 -12435.168,E2 -12435.168} C_VEL
LIN {X 0,Y 376.024,Z 232.644,A -85,B 0,C 180,E1 -12438.526,E2 -12438.526} C_VEL
LIN {X 0,Y 375.956,Z 232.652,A -85,B 0,C 180,E1 -12441.955,E2 -12441.955} C_VEL
LIN {X 0,Y 375.976,Z 232.651,A -85,B 0,C 180,E1 -12445.463,E2 -12445.463} C_VEL
LIN {X 0,Y 375.928,Z 232.65,A -85,B 0,C 180,E1 -12449.083,E2 -12449.083} C_VEL
LIN {X 0,Y 375.957,Z 232.652,A -85,B 0,C 180,E1 -12451.562,E2 -12451.562} C_VEL
LIN {X 0,Y 375.956,Z 232.656,A -85,B 0,C 180,E1 -12455.416,E2 -12455.416} C_VEL
LIN {X 0,Y 375.935,Z 232.663,A -85,B 0,C 180,E1 -12458.263,E2 -12458.263} C_VEL
LIN {X 0,Y 375.988,Z 232.709,A -85,B 0,C 180,E1 -12459.971,E2 -12459.971} C_VEL
LIN {X 0,Y 378.46,Z 244.567,A -85,B 0,C 180,E1 -12463.036,E2 -12463.036} C_VEL
LIN {X 0,Y 378.828,Z 246.682,A -85,B 0,C 180,E1 -12463.57,E2 -12463.57} C_VEL
LIN {X 0,Y 381.636,Z 258.107,A -85,B 0,C 180,E1 -12463.994,E2 -12463.994} C_VEL
LIN {X 0,Y 384.393,Z 272.784,A -85,B 0,C 180,E1 -12464.465,E2 -12464.465} C_VEL
LIN {X 0,Y 382.763,Z 355.18,A -85,B 0,C 180,E1 -12466.076,E2 -12466.076} C_VEL
LIN {X 0,Y 382.225,Z 369.162,A -85,B 0,C 180,E1 -12466.59,E2 -12466.59} C_VEL
LIN {X 0,Y 381.519,Z 381.554,A -85,B 0,C 180,E1 -12467.269,E2 -12467.269} C_VEL
LIN {X 0,Y 380.584,Z 393.855,A -85,B 0,C 180,E1 -12468.182,E2 -12468.182} C_VEL
LIN {X 0,Y 379.696,Z 404.604,A -85,B 0,C 180,E1 -12469.208,E2 -12469.208} C_VEL
LIN {X 0,Y 378.725,Z 414.401,A -85,B 0,C 180,E1 -12470.365,E2 -12470.365} C_VEL
LIN {X 0,Y 377.786,Z 422.857,A -85,B 0,C 180,E1 -12471.585,E2 -12471.585} C_VEL
LIN {X 0,Y 376.954,Z 431.082,A -85,B 0,C 180,E1 -12473.04,E2 -12473.04} C_VEL
LIN {X 0,Y 376.148,Z 438.289,A -85,B 0,C 180,E1 -12474.605,E2 -12474.605} C_VEL
LIN {X 0,Y 375.456,Z 445.125,A -85,B 0,C 180,E1 -12476.482,E2 -12476.482} C_VEL
LIN {X 0,Y 375.017,Z 450.23,A -85,B 0,C 180,E1 -12478.35,E2 -12478.35} C_VEL
LIN {X 0,Y 374.791,Z 452.885,A -85,B 0,C 180,E1 -12479.608,E2 -12479.608} C_VEL
LIN {X 0,Y 374.601,Z 454.832,A -85,B 0,C 180,E1 -12480.804,E2 -12480.804} C_VEL
LIN {X 0,Y 374.435,Z 456.275,A -85,B 0,C 180,E1 -12482.015,E2 -12482.015} C_VEL
LIN {X 0,Y 374.323,Z 457.223,A -85,B 0,C 180,E1 -12483.217,E2 -12483.217} C_VEL
LIN {X 0,Y 374.269,Z 457.628,A -85,B 0,C 180,E1 -12484.412,E2 -12484.412} C_VEL
LIN {X 0,Y 374.235,Z 457.582,A -85,B 0,C 180,E1 -12485.597,E2 -12485.597} C_VEL
LIN {X 0,Y 374.294,Z 456.926,A -85,B 0,C 180,E1 -12486.935,E2 -12486.935} C_VEL
LIN {X 0,Y 374.523,Z 454.56,A -85,B 0,C 180,E1 -12489.112,E2 -12489.112} C_VEL
LIN {X 0,Y 374.82,Z 451.428,A -85,B 0,C 180,E1 -12490.845,E2 -12490.845} C_VEL
LIN {X 0,Y 375.168,Z 446.362,A -85,B 0,C 180,E1 -12492.821,E2 -12492.821} C_VEL
LIN {X 0,Y 375.67,Z 440.544,A -85,B 0,C 180,E1 -12494.539,E2 -12494.539} C_VEL
LIN {X 0,Y 376.416,Z 432.828,A -85,B 0,C 180,E1 -12496.323,E2 -12496.323} C_VEL
LIN {X 0,Y 377.246,Z 424.185,A -85,B 0,C 180,E1 -12497.902,E2 -12497.902} C_VEL
LIN {X 0,Y 378.139,Z 414.805,A -85,B 0,C 180,E1 -12499.289,E2 -12499.289} C_VEL
LIN {X 0,Y 379.067,Z 404.369,A -85,B 0,C 180,E1 -12500.529,E2 -12500.529} C_VEL
LIN {X 0,Y 380.061,Z 392.659,A -85,B 0,C 180,E1 -12501.627,E2 -12501.627} C_VEL
LIN {X 0,Y 380.83,Z 380.55,A -85,B 0,C 180,E1 -12502.511,E2 -12502.511} C_VEL
LIN {X 0,Y 381.476,Z 367.649,A -85,B 0,C 180,E1 -12503.196,E2 -12503.196} C_VEL
LIN {X 0,Y 381.937,Z 354.667,A -85,B 0,C 180,E1 -12503.661,E2 -12503.661} C_VEL
LIN {X 0,Y 383.306,Z 270.687,A -85,B 0,C 180,E1 -12505.298,E2 -12505.298} C_VEL
LIN {X 0,Y 378.489,Z 246.519,A -85,B 0,C 180,E1 -12506.074,E2 -12506.074} C_VEL
LIN {X 0,Y 377.236,Z 237.652,A -85,B 0,C 180,E1 -12508.398,E2 -12508.398} C_VEL
LIN {X 0,Y 376.535,Z 234.046,A -85,B 0,C 180,E1 -12509.373,E2 -12509.373} C_VEL
LIN {X 0,Y 375.917,Z 232.949,A -85,B 0,C 180,E1 -12509.911,E2 -12509.911} C_VEL
LIN {X 0,Y 373.715,Z 232.935,A -85,B 0,C 180,E1 -12511.056,E2 -12511.056} C_VEL
LIN {X 0,Y 370.089,Z 233.493,A -85,B 0,C 180,E1 -12512.844,E2 -12512.844} C_VEL
LIN {X 0,Y 369.079,Z 233.52,A -85,B 0,C 180,E1 -12513.78,E2 -12513.78} C_VEL
LIN {X 0,Y 368.982,Z 233.52,A -85,B 0,C 180,E1 -12514.097,E2 -12514.097} C_VEL
LIN {X 0,Y 369.162,Z 233.497,A -85,B 0,C 180,E1 -12516.559,E2 -12516.559} C_VEL
LIN {X 0,Y 369.066,Z 233.514,A -85,B 0,C 180,E1 -12519.868,E2 -12519.868} C_VEL
LIN {X 0,Y 369.04,Z 233.519,A -85,B 0,C 180,E1 -12523.772,E2 -12523.772} C_VEL
LIN {X 0,Y 369.003,Z 233.523,A -85,B 0,C 180,E1 -12527.768,E2 -12527.768} C_VEL
LIN {X 0,Y 368.912,Z 233.529,A -85,B 0,C 180,E1 -12531.22,E2 -12531.22} C_VEL
LIN {X 0,Y 368.937,Z 233.525,A -85,B 0,C 180,E1 -12534.776,E2 -12534.776} C_VEL
LIN {X 0,Y 368.917,Z 233.529,A -85,B 0,C 180,E1 -12538.441,E2 -12538.441} C_VEL
LIN {X 0,Y 368.911,Z 233.529,A -85,B 0,C 180,E1 -12540.987,E2 -12540.987} C_VEL
LIN {X 0,Y 368.937,Z 233.525,A -85,B 0,C 180,E1 -12544.853,E2 -12544.853} C_VEL
LIN {X 0,Y 368.904,Z 233.53,A -85,B 0,C 180,E1 -12548.639,E2 -12548.639} C_VEL
LIN {X 0,Y 368.875,Z 233.538,A -85,B 0,C 180,E1 -12552.008,E2 -12552.008} C_VEL
LIN {X 0,Y 368.879,Z 233.533,A -85,B 0,C 180,E1 -12555.175,E2 -12555.175} C_VEL
LIN {X 0,Y 368.882,Z 233.537,A -85,B 0,C 180,E1 -12558.177,E2 -12558.177} C_VEL
LIN {X 0,Y 368.906,Z 233.53,A -85,B 0,C 180,E1 -12561.359,E2 -12561.359} C_VEL
LIN {X 0,Y 368.935,Z 233.526,A -85,B 0,C 180,E1 -12565.146,E2 -12565.146} C_VEL
LIN {X 0,Y 368.927,Z 233.527,A -85,B 0,C 180,E1 -12569.046,E2 -12569.046} C_VEL
LIN {X 0,Y 368.961,Z 233.523,A -85,B 0,C 180,E1 -12572.796,E2 -12572.796} C_VEL
LIN {X 0,Y 368.944,Z 233.53,A -85,B 0,C 180,E1 -12576.112,E2 -12576.112} C_VEL
LIN {X 0,Y 368.935,Z 233.531,A -85,B 0,C 180,E1 -12579.947,E2 -12579.947} C_VEL
LIN {X 0,Y 368.973,Z 233.522,A -85,B 0,C 180,E1 -12583.398,E2 -12583.398} C_VEL
LIN {X 0,Y 369.055,Z 233.512,A -85,B 0,C 180,E1 -12586.79,E2 -12586.79} C_VEL
LIN {X 0,Y 369.065,Z 233.515,A -85,B 0,C 180,E1 -12590.132,E2 -12590.132} C_VEL
LIN {X 0,Y 369.186,Z 233.499,A -85,B 0,C 180,E1 -12592.342,E2 -12592.342} C_VEL
LIN {X 0,Y 369.142,Z 233.503,A -85,B 0,C 180,E1 -12594.537,E2 -12594.537} C_VEL
LIN {X 0,Y 369.316,Z 233.481,A -85,B 0,C 180,E1 -12597.819,E2 -12597.819} C_VEL
LIN {X 0,Y 369.454,Z 233.466,A -85,B 0,C 180,E1 -12600,E2 -12600} C_VEL
LIN {X 0,Y 369.316,Z 233.483,A -85,B 0,C 180,E1 -12602.181,E2 -12602.181} C_VEL
LIN {X 0,Y 369.206,Z 233.495,A -85,B 0,C 180,E1 -12606.558,E2 -12606.558} C_VEL
LIN {X 0,Y 369.135,Z 233.502,A -85,B 0,C 180,E1 -12608.761,E2 -12608.761} C_VEL
LIN {X 0,Y 369.003,Z 233.522,A -85,B 0,C 180,E1 -12612.093,E2 -12612.093} C_VEL
LIN {X 0,Y 368.995,Z 233.519,A -85,B 0,C 180,E1 -12615.465,E2 -12615.465} C_VEL
LIN {X 0,Y 368.98,Z 233.521,A -85,B 0,C 180,E1 -12618.893,E2 -12618.893} C_VEL
LIN {X 0,Y 368.93,Z 233.532,A -85,B 0,C 180,E1 -12622.395,E2 -12622.395} C_VEL
LIN {X 0,Y 368.998,Z 233.521,A -85,B 0,C 180,E1 -12625.98,E2 -12625.98} C_VEL
LIN {X 0,Y 368.959,Z 233.525,A -85,B 0,C 180,E1 -12628.812,E2 -12628.812} C_VEL
LIN {X 0,Y 368.896,Z 233.535,A -85,B 0,C 180,E1 -12632.238,E2 -12632.238} C_VEL
LIN {X 0,Y 368.927,Z 233.527,A -85,B 0,C 180,E1 -12635.002,E2 -12635.002} C_VEL
LIN {X 0,Y 368.906,Z 233.533,A -85,B 0,C 180,E1 -12638.641,E2 -12638.641} C_VEL
LIN {X 0,Y 368.88,Z 233.535,A -85,B 0,C 180,E1 -12642.01,E2 -12642.01} C_VEL
LIN {X 0,Y 368.878,Z 233.533,A -85,B 0,C 180,E1 -12645.176,E2 -12645.176} C_VEL
LIN {X 0,Y 368.882,Z 233.536,A -85,B 0,C 180,E1 -12648.178,E2 -12648.178} C_VEL
LIN {X 0,Y 368.907,Z 233.529,A -85,B 0,C 180,E1 -12651.36,E2 -12651.36} C_VEL
LIN {X 0,Y 368.936,Z 233.526,A -85,B 0,C 180,E1 -12655.147,E2 -12655.147} C_VEL
LIN {X 0,Y 368.929,Z 233.532,A -85,B 0,C 180,E1 -12659.047,E2 -12659.047} C_VEL
LIN {X 0,Y 368.97,Z 233.568,A -85,B 0,C 180,E1 -12660.791,E2 -12660.791} C_VEL
LIN {X 0,Y 371.237,Z 244.497,A -85,B 0,C 180,E1 -12663.584,E2 -12663.584} C_VEL
LIN {X 0,Y 372.485,Z 252.188,A -85,B 0,C 180,E1 -12665.475,E2 -12665.475} C_VEL
LIN {X 0,Y 371.482,Z 263.207,A -85,B 0,C 180,E1 -12667.976,E2 -12667.976} C_VEL
LIN {X 0,Y 371.28,Z 265.917,A -85,B 0,C 180,E1 -12668.589,E2 -12668.589} C_VEL
LIN {X 0,Y 376.376,Z 298.249,A -85,B 0,C 180,E1 -12669.533,E2 -12669.533} C_VEL
LIN {X 0,Y 375.064,Z 374.241,A -85,B 0,C 180,E1 -12671.035,E2 -12671.035} C_VEL
LIN {X 0,Y 374.476,Z 387.38,A -85,B 0,C 180,E1 -12671.501,E2 -12671.501} C_VEL
LIN {X 0,Y 373.633,Z 400.621,A -85,B 0,C 180,E1 -12672.202,E2 -12672.202} C_VEL
LIN {X 0,Y 372.754,Z 411.762,A -85,B 0,C 180,E1 -12673.008,E2 -12673.008} C_VEL
LIN {X 0,Y 371.717,Z 423.369,A -85,B 0,C 180,E1 -12674.089,E2 -12674.089} C_VEL
LIN {X 0,Y 370.853,Z 433.699,A -85,B 0,C 180,E1 -12675.3,E2 -12675.3} C_VEL
LIN {X 0,Y 370.028,Z 442.38,A -85,B 0,C 180,E1 -12676.546,E2 -12676.546} C_VEL
LIN {X 0,Y 369.019,Z 451.628,A -85,B 0,C 180,E1 -12678.186,E2 -12678.186} C_VEL
LIN {X 0,Y 368.359,Z 459.065,A -85,B 0,C 180,E1 -12679.835,E2 -12679.835} C_VEL
LIN {X 0,Y 367.842,Z 465.898,A -85,B 0,C 180,E1 -12681.762,E2 -12681.762} C_VEL
LIN {X 0,Y 367.564,Z 470.396,A -85,B 0,C 180,E1 -12683.413,E2 -12683.413} C_VEL
LIN {X 0,Y 367.464,Z 472.766,A -85,B 0,C 180,E1 -12684.513,E2 -12684.513} C_VEL
LIN {X 0,Y 367.455,Z 474.703,A -85,B 0,C 180,E1 -12685.613,E2 -12685.613} C_VEL
LIN {X 0,Y 367.38,Z 476.207,A -85,B 0,C 180,E1 -12686.71,E2 -12686.71} C_VEL
LIN {X 0,Y 367.417,Z 477.916,A -85,B 0,C 180,E1 -12688.904,E2 -12688.904} C_VEL
LIN {X 0,Y 367.457,Z 478.185,A -85,B 0,C 180,E1 -12690,E2 -12690} C_VEL
LIN {X 0,Y 367.402,Z 478.049,A -85,B 0,C 180,E1 -12691.096,E2 -12691.096} C_VEL
LIN {X 0,Y 367.378,Z 476.518,A -85,B 0,C 180,E1 -12693.29,E2 -12693.29} C_VEL
LIN {X 0,Y 367.436,Z 475.161,A -85,B 0,C 180,E1 -12694.388,E2 -12694.388} C_VEL
LIN {X 0,Y 367.475,Z 472.355,A -85,B 0,C 180,E1 -12696.007,E2 -12696.007} C_VEL
LIN {X 0,Y 367.722,Z 468.4,A -85,B 0,C 180,E1 -12697.689,E2 -12697.689} C_VEL
LIN {X 0,Y 368.14,Z 463.377,A -85,B 0,C 180,E1 -12699.339,E2 -12699.339} C_VEL
LIN {X 0,Y 368.721,Z 457.076,A -85,B 0,C 180,E1 -12700.988,E2 -12700.988} C_VEL
LIN {X 0,Y 369.633,Z 449.203,A -85,B 0,C 180,E1 -12702.63,E2 -12702.63} C_VEL
LIN {X 0,Y 370.496,Z 441.182,A -85,B 0,C 180,E1 -12703.996,E2 -12703.996} C_VEL
LIN {X 0,Y 371.438,Z 431.409,A -85,B 0,C 180,E1 -12705.361,E2 -12705.361} C_VEL
LIN {X 0,Y 372.589,Z 420.554,A -85,B 0,C 180,E1 -12706.577,E2 -12706.577} C_VEL
LIN {X 0,Y 373.577,Z 409.963,A -85,B 0,C 180,E1 -12707.518,E2 -12707.518} C_VEL
LIN {X 0,Y 374.66,Z 397.244,A -85,B 0,C 180,E1 -12708.383,E2 -12708.383} C_VEL
LIN {X 0,Y 375.467,Z 384.538,A -85,B 0,C 180,E1 -12709.015,E2 -12709.015} C_VEL
LIN {X 0,Y 376.115,Z 370.899,A -85,B 0,C 180,E1 -12709.441,E2 -12709.441} C_VEL
LIN {X 0,Y 377.24,Z 297.203,A -85,B 0,C 180,E1 -12710.909,E2 -12710.909} C_VEL
LIN {X 0,Y 373.358,Z 273.49,A -85,B 0,C 180,E1 -12711.655,E2 -12711.655} C_VEL
LIN {X 0,Y 371.719,Z 265.002,A -85,B 0,C 180,E1 -12711.979,E2 -12711.979} C_VEL
LIN {X 0,Y 372.738,Z 253.715,A -85,B 0,C 180,E1 -12714.507,E2 -12714.507} C_VEL
LIN {X 0,Y 372.437,Z 250.245,A -85,B 0,C 180,E1 -12715.335,E2 -12715.335} C_VEL
LIN {X 0,Y 370.355,Z 239.604,A -85,B 0,C 180,E1 -12718.012,E2 -12718.012} C_VEL
LIN {X 0,Y 368.925,Z 233.532,A -85,B 0,C 180,E1 -12719.634,E2 -12719.634} C_VEL
LIN {X 0,Y 368.898,Z 233.537,A -85,B 0,C 180,E1 -12723.043,E2 -12723.043} C_VEL
LIN {X 0,Y 368.917,Z 233.53,A -85,B 0,C 180,E1 -12726.197,E2 -12726.197} C_VEL
LIN {X 0,Y 368.903,Z 233.534,A -85,B 0,C 180,E1 -12728.953,E2 -12728.953} C_VEL
LIN {X 0,Y 368.882,Z 233.533,A -85,B 0,C 180,E1 -12732.009,E2 -12732.009} C_VEL
LIN {X 0,Y 368.881,Z 233.535,A -85,B 0,C 180,E1 -12735.176,E2 -12735.176} C_VEL
LIN {X 0,Y 368.882,Z 233.53,A -85,B 0,C 180,E1 -12738.177,E2 -12738.177} C_VEL
LIN {X 0,Y 368.907,Z 233.529,A -85,B 0,C 180,E1 -12741.36,E2 -12741.36} C_VEL
LIN {X 0,Y 368.936,Z 233.524,A -85,B 0,C 180,E1 -12745.146,E2 -12745.146} C_VEL
LIN {X 0,Y 368.929,Z 233.524,A -85,B 0,C 180,E1 -12749.046,E2 -12749.046} C_VEL
LIN {X 0,Y 368.962,Z 233.519,A -85,B 0,C 180,E1 -12752.796,E2 -12752.796} C_VEL
LIN {X 0,Y 368.945,Z 233.523,A -85,B 0,C 180,E1 -12756.113,E2 -12756.113} C_VEL
LIN {X 0,Y 368.936,Z 233.525,A -85,B 0,C 180,E1 -12759.947,E2 -12759.947} C_VEL
LIN {X 0,Y 368.976,Z 233.523,A -85,B 0,C 180,E1 -12763.399,E2 -12763.399} C_VEL
LIN {X 0,Y 369.057,Z 233.507,A -85,B 0,C 180,E1 -12766.79,E2 -12766.79} C_VEL
LIN {X 0,Y 369.067,Z 233.505,A -85,B 0,C 180,E1 -12770.132,E2 -12770.132} C_VEL
LIN {X 0,Y 369.161,Z 233.498,A -85,B 0,C 180,E1 -12772.342,E2 -12772.342} C_VEL
LIN {X 0,Y 369.141,Z 233.499,A -85,B 0,C 180,E1 -12774.538,E2 -12774.538} C_VEL
LIN {X 0,Y 369.318,Z 233.479,A -85,B 0,C 180,E1 -12777.819,E2 -12777.819} C_VEL
LIN {X 0,Y 369.456,Z 233.454,A -85,B 0,C 180,E1 -12780,E2 -12780} C_VEL
LIN {X 0,Y 369.317,Z 233.48,A -85,B 0,C 180,E1 -12782.181,E2 -12782.181} C_VEL
LIN {X 0,Y 369.206,Z 233.497,A -85,B 0,C 180,E1 -12786.565,E2 -12786.565} C_VEL
LIN {X 0,Y 369.137,Z 233.5,A -85,B 0,C 180,E1 -12788.761,E2 -12788.761} C_VEL
LIN {X 0,Y 369.004,Z 233.514,A -85,B 0,C 180,E1 -12792.093,E2 -12792.093} C_VEL
LIN {X 0,Y 368.998,Z 233.517,A -85,B 0,C 180,E1 -12795.465,E2 -12795.465} C_VEL
LIN {X 0,Y 368.982,Z 233.523,A -85,B 0,C 180,E1 -12798.893,E2 -12798.893} C_VEL
LIN {X 0,Y 368.922,Z 233.532,A -85,B 0,C 180,E1 -12802.396,E2 -12802.396} C_VEL
LIN {X 0,Y 368.958,Z 233.526,A -85,B 0,C 180,E1 -12805.984,E2 -12805.984} C_VEL
LIN {X 0,Y 368.9,Z 233.528,A -85,B 0,C 180,E1 -12809.692,E2 -12809.692} C_VEL
LIN {X 0,Y 368.897,Z 233.535,A -85,B 0,C 180,E1 -12813.043,E2 -12813.043} C_VEL
LIN {X 0,Y 368.916,Z 233.538,A -85,B 0,C 180,E1 -12816.197,E2 -12816.197} C_VEL
LIN {X 0,Y 368.909,Z 233.535,A -85,B 0,C 180,E1 -12819.57,E2 -12819.57} C_VEL
LIN {X 0,Y 371.189,Z 244.177,A -85,B 0,C 180,E1 -12822.404,E2 -12822.404} C_VEL
LIN {X 0,Y 371.773,Z 247.109,A -85,B 0,C 180,E1 -12823.116,E2 -12823.116} C_VEL
LIN {X 0,Y 373.927,Z 254.054,A -85,B 0,C 180,E1 -12823.409,E2 -12823.409} C_VEL
LIN {X 0,Y 377.792,Z 272.881,A -85,B 0,C 180,E1 -12824.057,E2 -12824.057} C_VEL
LIN {X 0,Y 376.129,Z 354.763,A -85,B 0,C 180,E1 -12825.685,E2 -12825.685} C_VEL
LIN {X 0,Y 375.591,Z 368.429,A -85,B 0,C 180,E1 -12826.185,E2 -12826.185} C_VEL
LIN {X 0,Y 374.966,Z 379.425,A -85,B 0,C 180,E1 -12826.771,E2 -12826.771} C_VEL
LIN {X 0,Y 374.074,Z 391.447,A -85,B 0,C 180,E1 -12827.623,E2 -12827.623} C_VEL
LIN {X 0,Y 373.15,Z 401.91,A -85,B 0,C 180,E1 -12828.582,E2 -12828.582} C_VEL
LIN {X 0,Y 372.047,Z 413.023,A -85,B 0,C 180,E1 -12829.863,E2 -12829.863} C_VEL
LIN {X 0,Y 370.917,Z 423.003,A -85,B 0,C 180,E1 -12831.298,E2 -12831.298} C_VEL
LIN {X 0,Y 369.943,Z 431.984,A -85,B 0,C 180,E1 -12832.93,E2 -12832.93} C_VEL
LIN {X 0,Y 369.136,Z 438.881,A -85,B 0,C 180,E1 -12834.479,E2 -12834.479} C_VEL
LIN {X 0,Y 368.496,Z 444.67,A -85,B 0,C 180,E1 -12836.092,E2 -12836.092} C_VEL
LIN {X 0,Y 368.103,Z 449.193,A -85,B 0,C 180,E1 -12837.684,E2 -12837.684} C_VEL
LIN {X 0,Y 367.764,Z 452.761,A -85,B 0,C 180,E1 -12839.312,E2 -12839.312} C_VEL
LIN {X 0,Y 367.412,Z 455.967,A -85,B 0,C 180,E1 -12841.431,E2 -12841.431} C_VEL
LIN {X 0,Y 367.26,Z 457.081,A -85,B 0,C 180,E1 -12842.66,E2 -12842.66} C_VEL
LIN {X 0,Y 367.22,Z 457.787,A -85,B 0,C 180,E1 -12844.094,E2 -12844.094} C_VEL
LIN {X 0,Y 367.146,Z 457.508,A -85,B 0,C 180,E1 -12846.298,E2 -12846.298} C_VEL
LIN {X 0,Y 367.246,Z 456.712,A -85,B 0,C 180,E1 -12847.496,E2 -12847.496} C_VEL
LIN {X 0,Y 367.511,Z 454.135,A -85,B 0,C 180,E1 -12849.561,E2 -12849.561} C_VEL
LIN {X 0,Y 367.876,Z 450.06,A -85,B 0,C 180,E1 -12851.626,E2 -12851.626} C_VEL
LIN {X 0,Y 368.205,Z 445.327,A -85,B 0,C 180,E1 -12853.363,E2 -12853.363} C_VEL
LIN {X 0,Y 368.776,Z 439.227,A -85,B 0,C 180,E1 -12855.091,E2 -12855.091} C_VEL
LIN {X 0,Y 369.532,Z 431.569,A -85,B 0,C 180,E1 -12856.807,E2 -12856.807} C_VEL
LIN {X 0,Y 370.344,Z 423.733,A -85,B 0,C 180,E1 -12858.229,E2 -12858.229} C_VEL
LIN {X 0,Y 371.203,Z 415.184,A -85,B 0,C 180,E1 -12859.506,E2 -12859.506} C_VEL
LIN {X 0,Y 372.154,Z 404.86,A -85,B 0,C 180,E1 -12860.763,E2 -12860.763} C_VEL
LIN {X 0,Y 373.203,Z 393.197,A -85,B 0,C 180,E1 -12861.88,E2 -12861.88} C_VEL
LIN {X 0,Y 374,Z 381.186,A -85,B 0,C 180,E1 -12862.781,E2 -12862.781} C_VEL
LIN {X 0,Y 374.631,Z 368.714,A -85,B 0,C 180,E1 -12863.469,E2 -12863.469} C_VEL
LIN {X 0,Y 375.158,Z 355.399,A -85,B 0,C 180,E1 -12863.964,E2 -12863.964} C_VEL
LIN {X 0,Y 375.878,Z 319.818,A -85,B 0,C 180,E1 -12864.688,E2 -12864.688} C_VEL
LIN {X 0,Y 376.565,Z 271.379,A -85,B 0,C 180,E1 -12865.639,E2 -12865.639} C_VEL
LIN {X 0,Y 371.712,Z 247.828,A -85,B 0,C 180,E1 -12866.393,E2 -12866.393} C_VEL
LIN {X 0,Y 371.465,Z 246.794,A -85,B 0,C 180,E1 -12866.441,E2 -12866.441} C_VEL
LIN {X 0,Y 369.997,Z 237.6,A -85,B 0,C 180,E1 -12868.911,E2 -12868.911} C_VEL
LIN {X 0,Y 369.24,Z 233.487,A -85,B 0,C 180,E1 -12870.068,E2 -12870.068} C_VEL
LIN {X 0,Y 369.305,Z 233.483,A -85,B 0,C 180,E1 -12872.181,E2 -12872.181} C_VEL
LIN {X 0,Y 368.982,Z 233.52,A -85,B 0,C 180,E1 -12874.097,E2 -12874.097} C_VEL
LIN {X 0,Y 368.301,Z 233.606,A -85,B 0,C 180,E1 -12875.009,E2 -12875.009} C_VEL
LIN {X 0,Y 365.54,Z 233.952,A -85,B 0,C 180,E1 -12876.494,E2 -12876.494} C_VEL
LIN {X 0,Y 363.198,Z 234.246,A -85,B 0,C 180,E1 -12877.694,E2 -12877.694} C_VEL
LIN {X 0,Y 362.155,Z 234.372,A -85,B 0,C 180,E1 -12878.621,E2 -12878.621} C_VEL
LIN {X 0,Y 362.048,Z 234.383,A -85,B 0,C 180,E1 -12878.934,E2 -12878.934} C_VEL
LIN {X 0,Y 361.962,Z 234.395,A -85,B 0,C 180,E1 -12882.332,E2 -12882.332} C_VEL
LIN {X 0,Y 361.964,Z 234.394,A -85,B 0,C 180,E1 -12884.62,E2 -12884.62} C_VEL
LIN {X 0,Y 361.958,Z 234.398,A -85,B 0,C 180,E1 -12888.099,E2 -12888.099} C_VEL
LIN {X 0,Y 361.883,Z 234.408,A -85,B 0,C 180,E1 -12891.653,E2 -12891.653} C_VEL
LIN {X 0,Y 361.896,Z 234.404,A -85,B 0,C 180,E1 -12895.292,E2 -12895.292} C_VEL
LIN {X 0,Y 361.856,Z 234.408,A -85,B 0,C 180,E1 -12899.073,E2 -12899.073} C_VEL
LIN {X 0,Y 361.849,Z 234.408,A -85,B 0,C 180,E1 -12902.944,E2 -12902.944} C_VEL
LIN {X 0,Y 361.868,Z 234.409,A -85,B 0,C 180,E1 -12905.636,E2 -12905.636} C_VEL
LIN {X 0,Y 361.865,Z 234.406,A -85,B 0,C 180,E1 -12909.025,E2 -12909.025} C_VEL
LIN {X 0,Y 361.834,Z 234.41,A -85,B 0,C 180,E1 -12912.829,E2 -12912.829} C_VEL
LIN {X 0,Y 361.818,Z 234.418,A -85,B 0,C 180,E1 -12915.946,E2 -12915.946} C_VEL
LIN {X 0,Y 361.834,Z 234.411,A -85,B 0,C 180,E1 -12919.244,E2 -12919.244} C_VEL
LIN {X 0,Y 361.862,Z 234.407,A -85,B 0,C 180,E1 -12922.777,E2 -12922.777} C_VEL
LIN {X 0,Y 361.853,Z 234.411,A -85,B 0,C 180,E1 -12925.719,E2 -12925.719} C_VEL
LIN {X 0,Y 361.871,Z 234.408,A -85,B 0,C 180,E1 -12929.672,E2 -12929.672} C_VEL
LIN {X 0,Y 361.952,Z 234.397,A -85,B 0,C 180,E1 -12933.475,E2 -12933.475} C_VEL
LIN {X 0,Y 361.888,Z 234.403,A -85,B 0,C 180,E1 -12937.144,E2 -12937.144} C_VEL
LIN {X 0,Y 361.91,Z 234.402,A -85,B 0,C 180,E1 -12940.723,E2 -12940.723} C_VEL
LIN {X 0,Y 361.93,Z 234.398,A -85,B 0,C 180,E1 -12943.066,E2 -12943.066} C_VEL
LIN {X 0,Y 361.996,Z 234.392,A -85,B 0,C 180,E1 -12946.528,E2 -12946.528} C_VEL
